LIN {X 0,Y 469.729,Z 273.756,A -85,B 0,C 180,E1 -7607.149,E2 -7607.149} C_VEL
LIN {X 0,Y 469.923,Z 277.249,A -85,B 0,C 180,E1 -7608.848,E2 -7608.848} C_VEL
LIN {X 0,Y 469.592,Z 283.298,A -85,B 0,C 180,E1 -7611.619,E2 -7611.619} C_VEL
LIN {X 0,Y 469.198,Z 289.323,A -85,B 0,C 180,E1 -7614.255,E2 -7614.255} C_VEL
LIN {X 0,Y 468.777,Z 296.664,A -85,B 0,C 180,E1 -7617.335,E2 -7617.335} C_VEL
LIN {X 0,Y 468.436,Z 304.481,A -85,B 0,C 180,E1 -7620.479,E2 -7620.479} C_VEL
LIN {X 0,Y 468.052,Z 312.815,A -85,B 0,C 180,E1 -7623.707,E2 -7623.707} C_VEL
LIN {X 0,Y 467.727,Z 321.729,A -85,B 0,C 180,E1 -7627.003,E2 -7627.003} C_VEL
LIN {X 0,Y 467.618,Z 324.914,A -85,B 0,C 180,E1 -7628.178,E2 -7628.178} C_VEL
LIN {X 0,Y 472.483,Z 344.192,A -85,B 0,C 180,E1 -7628.855,E2 -7628.855} C_VEL
LIN {X 0,Y 473.831,Z 350.735,A -85,B 0,C 180,E1 -7629.122,E2 -7629.122} C_VEL
LIN {X 0,Y 473.198,Z 365.39,A -85,B 0,C 180,E1 -7629.679,E2 -7629.679} C_VEL
LIN {X 0,Y 472.423,Z 380.522,A -85,B 0,C 180,E1 -7630.444,E2 -7630.444} C_VEL
LIN {X 0,Y 471.631,Z 394.097,A -85,B 0,C 180,E1 -7631.314,E2 -7631.314} C_VEL
LIN {X 0,Y 470.815,Z 406.65,A -85,B 0,C 180,E1 -7632.293,E2 -7632.293} C_VEL
LIN {X 0,Y 469.962,Z 419.312,A -85,B 0,C 180,E1 -7633.493,E2 -7633.493} C_VEL
LIN {X 0,Y 469.169,Z 430.767,A -85,B 0,C 180,E1 -7634.803,E2 -7634.803} C_VEL
LIN {X 0,Y 468.498,Z 440.435,A -85,B 0,C 180,E1 -7636.112,E2 -7636.112} C_VEL
LIN {X 0,Y 467.896,Z 449.138,A -85,B 0,C 180,E1 -7637.508,E2 -7637.508} C_VEL
LIN {X 0,Y 467.494,Z 457.77,A -85,B 0,C 180,E1 -7639.169,E2 -7639.169} C_VEL
LIN {X 0,Y 467.07,Z 465.123,A -85,B 0,C 180,E1 -7640.909,E2 -7640.909} C_VEL
LIN {X 0,Y 466.83,Z 470.949,A -85,B 0,C 180,E1 -7642.648,E2 -7642.648} C_VEL
LIN {X 0,Y 466.753,Z 474.383,A -85,B 0,C 180,E1 -7643.95,E2 -7643.95} C_VEL
LIN {X 0,Y 466.619,Z 477.892,A -85,B 0,C 180,E1 -7645.681,E2 -7645.681} C_VEL
LIN {X 0,Y 466.638,Z 480.197,A -85,B 0,C 180,E1 -7647.41,E2 -7647.41} C_VEL
LIN {X 0,Y 466.586,Z 481.352,A -85,B 0,C 180,E1 -7649.137,E2 -7649.137} C_VEL
LIN {X 0,Y 466.586,Z 481.35,A -85,B 0,C 180,E1 -7650.863,E2 -7650.863} C_VEL
LIN {X 0,Y 466.638,Z 480.191,A -85,B 0,C 180,E1 -7652.59,E2 -7652.59} C_VEL
LIN {X 0,Y 466.619,Z 477.886,A -85,B 0,C 180,E1 -7654.319,E2 -7654.319} C_VEL
LIN {X 0,Y 466.768,Z 474.383,A -85,B 0,C 180,E1 -7656.05,E2 -7656.05} C_VEL
LIN {X 0,Y 466.896,Z 469.596,A -85,B 0,C 180,E1 -7657.786,E2 -7657.786} C_VEL
LIN {X 0,Y 467.133,Z 463.399,A -85,B 0,C 180,E1 -7659.526,E2 -7659.526} C_VEL
LIN {X 0,Y 467.614,Z 455.624,A -85,B 0,C 180,E1 -7661.267,E2 -7661.267} C_VEL
LIN {X 0,Y 468.03,Z 447.084,A -85,B 0,C 180,E1 -7662.838,E2 -7662.838} C_VEL
LIN {X 0,Y 468.71,Z 437.348,A -85,B 0,C 180,E1 -7664.324,E2 -7664.324} C_VEL
LIN {X 0,Y 469.341,Z 427.143,A -85,B 0,C 180,E1 -7665.637,E2 -7665.637} C_VEL
LIN {X 0,Y 470.179,Z 415.078,A -85,B 0,C 180,E1 -7666.935,E2 -7666.935} C_VEL
LIN {X 0,Y 471.028,Z 402.621,A -85,B 0,C 180,E1 -7668.035,E2 -7668.035} C_VEL
LIN {X 0,Y 471.897,Z 389.15,A -85,B 0,C 180,E1 -7669.013,E2 -7669.013} C_VEL
LIN {X 0,Y 472.698,Z 375.343,A -85,B 0,C 180,E1 -7669.827,E2 -7669.827} C_VEL
LIN {X 0,Y 473.369,Z 360.123,A -85,B 0,C 180,E1 -7670.532,E2 -7670.532} C_VEL
LIN {X 0,Y 473.644,Z 349.558,A -85,B 0,C 180,E1 -7670.919,E2 -7670.919} C_VEL
LIN {X 0,Y 469.716,Z 332.966,A -85,B 0,C 180,E1 -7671.556,E2 -7671.556} C_VEL
LIN {X 0,Y 467.579,Z 324.175,A -85,B 0,C 180,E1 -7671.844,E2 -7671.844} C_VEL
LIN {X 0,Y 467.838,Z 314.394,A -85,B 0,C 180,E1 -7675.275,E2 -7675.275} C_VEL
LIN {X 0,Y 468.108,Z 306.24,A -85,B 0,C 180,E1 -7678.225,E2 -7678.225} C_VEL
LIN {X 0,Y 468.385,Z 298.351,A -85,B 0,C 180,E1 -7681.211,E2 -7681.211} C_VEL
LIN {X 0,Y 468.622,Z 292.205,A -85,B 0,C 180,E1 -7683.704,E2 -7683.704} C_VEL
LIN {X 0,Y 469.09,Z 285.23,A -85,B 0,C 180,E1 -7686.819,E2 -7686.819} C_VEL
LIN {X 0,Y 469.452,Z 281.021,A -85,B 0,C 180,E1 -7688.96,E2 -7688.96} C_VEL
LIN {X 0,Y 469.801,Z 277.325,A -85,B 0,C 180,E1 -7691.164,E2 -7691.164} C_VEL
LIN {X 0,Y 469.823,Z 275.034,A -85,B 0,C 180,E1 -7692.863,E2 -7692.863} C_VEL
LIN {X 0,Y 469.444,Z 272.713,A -85,B 0,C 180,E1 -7695.281,E2 -7695.281} C_VEL
LIN {X 0,Y 469.093,Z 271.43,A -85,B 0,C 180,E1 -7697.609,E2 -7697.609} C_VEL
LIN {X 0,Y 468.597,Z 271.032,A -85,B 0,C 180,E1 -7699.898,E2 -7699.898} C_VEL
LIN {X 0,Y 468.189,Z 271.444,A -85,B 0,C 180,E1 -7703.099,E2 -7703.099} C_VEL
LIN {X 0,Y 467.827,Z 272.613,A -85,B 0,C 180,E1 -7706.232,E2 -7706.232} C_VEL
LIN {X 0,Y 467.602,Z 274.182,A -85,B 0,C 180,E1 -7709.269,E2 -7709.269} C_VEL
LIN {X 0,Y 467.434,Z 276.177,A -85,B 0,C 180,E1 -7712.509,E2 -7712.509} C_VEL
LIN {X 0,Y 467.341,Z 277.655,A -85,B 0,C 180,E1 -7714.672,E2 -7714.672} C_VEL
LIN {X 0,Y 472.477,Z 293.108,A -85,B 0,C 180,E1 -7715.363,E2 -7715.363} C_VEL
LIN {X 0,Y 473.121,Z 296.754,A -85,B 0,C 180,E1 -7715.523,E2 -7715.523} C_VEL
LIN {X 0,Y 472.61,Z 311.746,A -85,B 0,C 180,E1 -7716.13,E2 -7716.13} C_VEL
LIN {X 0,Y 471.958,Z 326.057,A -85,B 0,C 180,E1 -7716.874,E2 -7716.874} C_VEL
LIN {X 0,Y 471.281,Z 339.483,A -85,B 0,C 180,E1 -7717.746,E2 -7717.746} C_VEL
LIN {X 0,Y 470.652,Z 351.07,A -85,B 0,C 180,E1 -7718.655,E2 -7718.655} C_VEL
LIN {X 0,Y 469.879,Z 364.056,A -85,B 0,C 180,E1 -7719.879,E2 -7719.879} C_VEL
LIN {X 0,Y 469.205,Z 375.809,A -85,B 0,C 180,E1 -7721.214,E2 -7721.214} C_VEL
LIN {X 0,Y 468.589,Z 385.608,A -85,B 0,C 180,E1 -7722.545,E2 -7722.545} C_VEL
LIN {X 0,Y 468.037,Z 395.102,A -85,B 0,C 180,E1 -7724.092,E2 -7724.092} C_VEL
LIN {X 0,Y 467.622,Z 402.939,A -85,B 0,C 180,E1 -7725.642,E2 -7725.642} C_VEL
LIN {X 0,Y 467.278,Z 410.166,A -85,B 0,C 180,E1 -7727.404,E2 -7727.404} C_VEL
LIN {X 0,Y 467.044,Z 415.784,A -85,B 0,C 180,E1 -7729.158,E2 -7729.158} C_VEL
LIN {X 0,Y 466.851,Z 419.086,A -85,B 0,C 180,E1 -7730.468,E2 -7730.468} C_VEL
LIN {X 0,Y 466.794,Z 422.271,A -85,B 0,C 180,E1 -7732.212,E2 -7732.212} C_VEL
LIN {X 0,Y 466.795,Z 424.199,A -85,B 0,C 180,E1 -7733.951,E2 -7733.951} C_VEL
LIN {X 0,Y 466.728,Z 424.95,A -85,B 0,C 180,E1 -7735.682,E2 -7735.682} C_VEL
LIN {X 0,Y 466.782,Z 424.534,A -85,B 0,C 180,E1 -7737.411,E2 -7737.411} C_VEL
LIN {X 0,Y 466.625,Z 422.981,A -85,B 0,C 180,E1 -7739.137,E2 -7739.137} C_VEL
LIN {X 0,Y 466.648,Z 420.238,A -85,B 0,C 180,E1 -7740.863,E2 -7740.863} C_VEL
LIN {X 0,Y 466.881,Z 416.228,A -85,B 0,C 180,E1 -7742.589,E2 -7742.589} C_VEL
LIN {X 0,Y 467.22,Z 410.87,A -85,B 0,C 180,E1 -7744.314,E2 -7744.314} C_VEL
LIN {X 0,Y 467.375,Z 404.075,A -85,B 0,C 180,E1 -7746.042,E2 -7746.042} C_VEL
LIN {X 0,Y 467.914,Z 395.592,A -85,B 0,C 180,E1 -7747.769,E2 -7747.769} C_VEL
LIN {X 0,Y 468.452,Z 386.549,A -85,B 0,C 180,E1 -7749.281,E2 -7749.281} C_VEL
LIN {X 0,Y 469.134,Z 375.671,A -85,B 0,C 180,E1 -7750.793,E2 -7750.793} C_VEL
LIN {X 0,Y 469.839,Z 364.496,A -85,B 0,C 180,E1 -7752.088,E2 -7752.088} C_VEL
LIN {X 0,Y 470.568,Z 352.274,A -85,B 0,C 180,E1 -7753.275,E2 -7753.275} C_VEL
LIN {X 0,Y 471.254,Z 339.027,A -85,B 0,C 180,E1 -7754.346,E2 -7754.346} C_VEL
LIN {X 0,Y 471.989,Z 325.833,A -85,B 0,C 180,E1 -7755.215,E2 -7755.215} C_VEL
LIN {X 0,Y 472.684,Z 310.816,A -85,B 0,C 180,E1 -7756.009,E2 -7756.009} C_VEL
LIN {X 0,Y 473.121,Z 295.089,A -85,B 0,C 180,E1 -7756.644,E2 -7756.644} C_VEL
LIN {X 0,Y 468.818,Z 279.993,A -85,B 0,C 180,E1 -7757.279,E2 -7757.279} C_VEL
LIN {X 0,Y 466.857,Z 273.316,A -85,B 0,C 180,E1 -7757.523,E2 -7757.523} C_VEL
LIN {X 0,Y 466.872,Z 270.616,A -85,B 0,C 180,E1 -7760.257,E2 -7760.257} C_VEL
LIN {X 0,Y 466.934,Z 267.582,A -85,B 0,C 180,E1 -7763.344,E2 -7763.344} C_VEL
LIN {X 0,Y 466.986,Z 265.148,A -85,B 0,C 180,E1 -7765.877,E2 -7765.877} C_VEL
LIN {X 0,Y 467.008,Z 262.347,A -85,B 0,C 180,E1 -7768.788,E2 -7768.788} C_VEL
LIN {X 0,Y 466.989,Z 261.962,A -85,B 0,C 180,E1 -7769.205,E2 -7769.205} C_VEL
LIN {X 0,Y 467.278,Z 261.908,A -85,B 0,C 180,E1 -7771.764,E2 -7771.764} C_VEL
LIN {X 0,Y 467.535,Z 261.872,A -85,B 0,C 180,E1 -7774.835,E2 -7774.835} C_VEL
LIN {X 0,Y 467.566,Z 261.867,A -85,B 0,C 180,E1 -7778.045,E2 -7778.045} C_VEL
LIN {X 0,Y 467.578,Z 261.868,A -85,B 0,C 180,E1 -7781.276,E2 -7781.276} C_VEL
LIN {X 0,Y 467.549,Z 261.868,A -85,B 0,C 180,E1 -7783.82,E2 -7783.82} C_VEL
LIN {X 0,Y 467.558,Z 261.87,A -85,B 0,C 180,E1 -7786.255,E2 -7786.255} C_VEL
LIN {X 0,Y 467.582,Z 261.867,A -85,B 0,C 180,E1 -7788.723,E2 -7788.723} C_VEL
LIN {X 0,Y 467.568,Z 261.867,A -85,B 0,C 180,E1 -7791.955,E2 -7791.955} C_VEL
LIN {X 0,Y 467.562,Z 261.871,A -85,B 0,C 180,E1 -7795.167,E2 -7795.167} C_VEL
LIN {X 0,Y 467.586,Z 261.866,A -85,B 0,C 180,E1 -7798.26,E2 -7798.26} C_VEL
LIN {X 0,Y 467.579,Z 261.868,A -85,B 0,C 180,E1 -7801.25,E2 -7801.25} C_VEL
LIN {X 0,Y 467.59,Z 261.865,A -85,B 0,C 180,E1 -7804.159,E2 -7804.159} C_VEL
LIN {X 0,Y 467.579,Z 261.867,A -85,B 0,C 180,E1 -7806.996,E2 -7806.996} C_VEL
LIN {X 0,Y 467.609,Z 261.862,A -85,B 0,C 180,E1 -7809.599,E2 -7809.599} C_VEL
LIN {X 0,Y 466.981,Z 261.943,A -85,B 0,C 180,E1 -7810.318,E2 -7810.318} C_VEL
LIN {X 0,Y 464.118,Z 262.299,A -85,B 0,C 180,E1 -7811.485,E2 -7811.485} C_VEL
LIN {X 0,Y 461.677,Z 262.603,A -85,B 0,C 180,E1 -7812.426,E2 -7812.426} C_VEL
LIN {X 0,Y 460.64,Z 262.731,A -85,B 0,C 180,E1 -7813.154,E2 -7813.154} C_VEL
LIN {X 0,Y 460.563,Z 262.74,A -85,B 0,C 180,E1 -7813.4,E2 -7813.4} C_VEL
LIN {X 0,Y 460.555,Z 262.742,A -85,B 0,C 180,E1 -7815.868,E2 -7815.868} C_VEL
LIN {X 0,Y 460.613,Z 262.734,A -85,B 0,C 180,E1 -7818.559,E2 -7818.559} C_VEL
LIN {X 0,Y 460.67,Z 262.728,A -85,B 0,C 180,E1 -7822.108,E2 -7822.108} C_VEL
LIN {X 0,Y 460.68,Z 262.724,A -85,B 0,C 180,E1 -7824.748,E2 -7824.748} C_VEL
LIN {X 0,Y 460.795,Z 262.713,A -85,B 0,C 180,E1 -7827.377,E2 -7827.377} C_VEL
LIN {X 0,Y 460.853,Z 262.706,A -85,B 0,C 180,E1 -7830,E2 -7830} C_VEL
LIN {X 0,Y 460.795,Z 262.71,A -85,B 0,C 180,E1 -7832.623,E2 -7832.623} C_VEL
LIN {X 0,Y 460.69,Z 262.727,A -85,B 0,C 180,E1 -7836.13,E2 -7836.13} C_VEL
LIN {X 0,Y 460.622,Z 262.731,A -85,B 0,C 180,E1 -7838.776,E2 -7838.776} C_VEL
LIN {X 0,Y 460.617,Z 262.735,A -85,B 0,C 180,E1 -7842.445,E2 -7842.445} C_VEL
LIN {X 0,Y 460.604,Z 262.735,A -85,B 0,C 180,E1 -7845.998,E2 -7845.998} C_VEL
LIN {X 0,Y 460.572,Z 262.74,A -85,B 0,C 180,E1 -7849.616,E2 -7849.616} C_VEL
LIN {X 0,Y 460.514,Z 262.744,A -85,B 0,C 180,E1 -7852.429,E2 -7852.429} C_VEL
LIN {X 0,Y 460.572,Z 262.741,A -85,B 0,C 180,E1 -7855.802,E2 -7855.802} C_VEL
LIN {X 0,Y 460.554,Z 262.741,A -85,B 0,C 180,E1 -7858.233,E2 -7858.233} C_VEL
LIN {X 0,Y 460.523,Z 262.746,A -85,B 0,C 180,E1 -7861.283,E2 -7861.283} C_VEL
LIN {X 0,Y 460.534,Z 262.744,A -85,B 0,C 180,E1 -7864.505,E2 -7864.505} C_VEL
LIN {X 0,Y 460.502,Z 262.748,A -85,B 0,C 180,E1 -7867.623,E2 -7867.623} C_VEL
LIN {X 0,Y 460.519,Z 262.747,A -85,B 0,C 180,E1 -7871.013,E2 -7871.013} C_VEL
LIN {X 0,Y 460.515,Z 262.748,A -85,B 0,C 180,E1 -7874.589,E2 -7874.589} C_VEL
LIN {X 0,Y 460.527,Z 262.745,A -85,B 0,C 180,E1 -7877.819,E2 -7877.819} C_VEL
LIN {X 0,Y 460.549,Z 262.742,A -85,B 0,C 180,E1 -7881.102,E2 -7881.102} C_VEL
LIN {X 0,Y 460.512,Z 262.747,A -85,B 0,C 180,E1 -7884.554,E2 -7884.554} C_VEL
LIN {X 0,Y 460.534,Z 262.743,A -85,B 0,C 180,E1 -7887.716,E2 -7887.716} C_VEL
LIN {X 0,Y 460.544,Z 262.744,A -85,B 0,C 180,E1 -7890.769,E2 -7890.769} C_VEL
LIN {X 0,Y 460.547,Z 262.74,A -85,B 0,C 180,E1 -7893.733,E2 -7893.733} C_VEL
LIN {X 0,Y 460.549,Z 262.743,A -85,B 0,C 180,E1 -7896.624,E2 -7896.624} C_VEL
LIN {X 0,Y 460.555,Z 262.74,A -85,B 0,C 180,E1 -7899.453,E2 -7899.453} C_VEL
LIN {X 0,Y 460.552,Z 262.744,A -85,B 0,C 180,E1 -7902.23,E2 -7902.23} C_VEL
LIN {X 0,Y 460.567,Z 262.741,A -85,B 0,C 180,E1 -7904.965,E2 -7904.965} C_VEL
LIN {X 0,Y 460.616,Z 262.734,A -85,B 0,C 180,E1 -7908.559,E2 -7908.559} C_VEL
LIN {X 0,Y 460.623,Z 262.733,A -85,B 0,C 180,E1 -7911.224,E2 -7911.224} C_VEL
LIN {X 0,Y 460.675,Z 262.727,A -85,B 0,C 180,E1 -7913.869,E2 -7913.869} C_VEL
LIN {X 0,Y 460.797,Z 262.713,A -85,B 0,C 180,E1 -7917.377,E2 -7917.377} C_VEL
LIN {X 0,Y 460.853,Z 262.706,A -85,B 0,C 180,E1 -7920,E2 -7920} C_VEL
LIN {X 0,Y 460.804,Z 262.71,A -85,B 0,C 180,E1 -7922.622,E2 -7922.622} C_VEL
LIN {X 0,Y 460.687,Z 262.728,A -85,B 0,C 180,E1 -7926.13,E2 -7926.13} C_VEL
LIN {X 0,Y 460.614,Z 262.733,A -85,B 0,C 180,E1 -7928.776,E2 -7928.776} C_VEL
LIN {X 0,Y 460.618,Z 262.734,A -85,B 0,C 180,E1 -7932.445,E2 -7932.445} C_VEL
LIN {X 0,Y 460.604,Z 262.735,A -85,B 0,C 180,E1 -7935.997,E2 -7935.997} C_VEL
LIN {X 0,Y 460.572,Z 262.741,A -85,B 0,C 180,E1 -7939.615,E2 -7939.615} C_VEL
LIN {X 0,Y 460.514,Z 262.745,A -85,B 0,C 180,E1 -7942.428,E2 -7942.428} C_VEL
LIN {X 0,Y 460.551,Z 262.744,A -85,B 0,C 180,E1 -7945.796,E2 -7945.796} C_VEL
LIN {X 0,Y 460.517,Z 262.744,A -85,B 0,C 180,E1 -7948.235,E2 -7948.235} C_VEL
LIN {X 0,Y 460.522,Z 262.746,A -85,B 0,C 180,E1 -7951.282,E2 -7951.282} C_VEL
LIN {X 0,Y 460.533,Z 262.744,A -85,B 0,C 180,E1 -7954.505,E2 -7954.505} C_VEL
LIN {X 0,Y 460.503,Z 262.746,A -85,B 0,C 180,E1 -7957.623,E2 -7957.623} C_VEL
LIN {X 0,Y 460.557,Z 262.915,A -85,B 0,C 180,E1 -7960.393,E2 -7960.393} C_VEL
LIN {X 0,Y 461.469,Z 267.969,A -85,B 0,C 180,E1 -7963.262,E2 -7963.262} C_VEL
LIN {X 0,Y 462.516,Z 273.431,A -85,B 0,C 180,E1 -7966.2,E2 -7966.2} C_VEL
LIN {X 0,Y 462.968,Z 277.166,A -85,B 0,C 180,E1 -7968.092,E2 -7968.092} C_VEL
LIN {X 0,Y 462.775,Z 281.979,A -85,B 0,C 180,E1 -7970.369,E2 -7970.369} C_VEL
LIN {X 0,Y 462.348,Z 289.228,A -85,B 0,C 180,E1 -7973.642,E2 -7973.642} C_VEL
LIN {X 0,Y 461.867,Z 296.621,A -85,B 0,C 180,E1 -7976.815,E2 -7976.815} C_VEL
LIN {X 0,Y 461.448,Z 304.97,A -85,B 0,C 180,E1 -7980.242,E2 -7980.242} C_VEL
LIN {X 0,Y 461.065,Z 312.637,A -85,B 0,C 180,E1 -7983.277,E2 -7983.277} C_VEL
LIN {X 0,Y 460.696,Z 321.458,A -85,B 0,C 180,E1 -7986.632,E2 -7986.632} C_VEL
LIN {X 0,Y 460.593,Z 324.594,A -85,B 0,C 180,E1 -7987.808,E2 -7987.808} C_VEL
LIN {X 0,Y 465.546,Z 344.217,A -85,B 0,C 180,E1 -7988.53,E2 -7988.53} C_VEL
LIN {X 0,Y 467.098,Z 351.971,A -85,B 0,C 180,E1 -7988.86,E2 -7988.86} C_VEL
LIN {X 0,Y 466.496,Z 365.604,A -85,B 0,C 180,E1 -7989.399,E2 -7989.399} C_VEL
LIN {X 0,Y 465.674,Z 380.141,A -85,B 0,C 180,E1 -7990.149,E2 -7990.149} C_VEL
LIN {X 0,Y 464.826,Z 393.687,A -85,B 0,C 180,E1 -7991.03,E2 -7991.03} C_VEL
LIN {X 0,Y 463.889,Z 407.452,A -85,B 0,C 180,E1 -7992.134,E2 -7992.134} C_VEL
LIN {X 0,Y 462.997,Z 419.97,A -85,B 0,C 180,E1 -7993.351,E2 -7993.351} C_VEL
LIN {X 0,Y 462.24,Z 430.537,A -85,B 0,C 180,E1 -7994.569,E2 -7994.569} C_VEL
LIN {X 0,Y 461.537,Z 440.328,A -85,B 0,C 180,E1 -7995.898,E2 -7995.898} C_VEL
LIN {X 0,Y 460.882,Z 449.651,A -85,B 0,C 180,E1 -7997.405,E2 -7997.405} C_VEL
LIN {X 0,Y 460.482,Z 457.77,A -85,B 0,C 180,E1 -7999.002,E2 -7999.002} C_VEL
LIN {X 0,Y 460.008,Z 465.124,A -85,B 0,C 180,E1 -8000.769,E2 -8000.769} C_VEL
LIN {X 0,Y 459.775,Z 470.95,A -85,B 0,C 180,E1 -8002.534,E2 -8002.534} C_VEL
LIN {X 0,Y 459.654,Z 474.382,A -85,B 0,C 180,E1 -8003.856,E2 -8003.856} C_VEL
LIN {X 0,Y 459.538,Z 477.892,A -85,B 0,C 180,E1 -8005.614,E2 -8005.614} C_VEL
LIN {X 0,Y 459.56,Z 480.197,A -85,B 0,C 180,E1 -8007.37,E2 -8007.37} C_VEL
LIN {X 0,Y 459.491,Z 481.352,A -85,B 0,C 180,E1 -8009.124,E2 -8009.124} C_VEL
LIN {X 0,Y 459.491,Z 481.35,A -85,B 0,C 180,E1 -8010.876,E2 -8010.876} C_VEL
LIN {X 0,Y 459.56,Z 480.191,A -85,B 0,C 180,E1 -8012.63,E2 -8012.63} C_VEL
LIN {X 0,Y 459.538,Z 477.886,A -85,B 0,C 180,E1 -8014.386,E2 -8014.386} C_VEL
LIN {X 0,Y 459.696,Z 474.383,A -85,B 0,C 180,E1 -8016.143,E2 -8016.143} C_VEL
LIN {X 0,Y 459.826,Z 469.595,A -85,B 0,C 180,E1 -8017.907,E2 -8017.907} C_VEL
LIN {X 0,Y 460.09,Z 463.397,A -85,B 0,C 180,E1 -8019.673,E2 -8019.673} C_VEL
LIN {X 0,Y 460.609,Z 455.621,A -85,B 0,C 180,E1 -8021.441,E2 -8021.441} C_VEL
LIN {X 0,Y 461.034,Z 447.195,A -85,B 0,C 180,E1 -8023.014,E2 -8023.014} C_VEL
LIN {X 0,Y 461.749,Z 437.152,A -85,B 0,C 180,E1 -8024.545,E2 -8024.545} C_VEL
LIN {X 0,Y 462.434,Z 426.739,A -85,B 0,C 180,E1 -8025.876,E2 -8025.876} C_VEL
LIN {X 0,Y 463.221,Z 415.491,A -85,B 0,C 180,E1 -8027.092,E2 -8027.092} C_VEL
LIN {X 0,Y 464.096,Z 403.283,A -85,B 0,C 180,E1 -8028.2,E2 -8028.2} C_VEL
LIN {X 0,Y 465.003,Z 390.115,A -85,B 0,C 180,E1 -8029.192,E2 -8029.192} C_VEL
LIN {X 0,Y 465.922,Z 375.728,A -85,B 0,C 180,E1 -8030.07,E2 -8030.07} C_VEL
LIN {X 0,Y 466.669,Z 360.221,A -85,B 0,C 180,E1 -8030.813,E2 -8030.813} C_VEL
LIN {X 0,Y 466.883,Z 350.717,A -85,B 0,C 180,E1 -8031.179,E2 -8031.179} C_VEL
LIN {X 0,Y 463.094,Z 334.414,A -85,B 0,C 180,E1 -8031.846,E2 -8031.846} C_VEL
LIN {X 0,Y 460.522,Z 323.542,A -85,B 0,C 180,E1 -8032.224,E2 -8032.224} C_VEL
LIN {X 0,Y 460.849,Z 313.364,A -85,B 0,C 180,E1 -8035.874,E2 -8035.874} C_VEL
LIN {X 0,Y 461.149,Z 304.471,A -85,B 0,C 180,E1 -8039.189,E2 -8039.189} C_VEL
LIN {X 0,Y 461.373,Z 298.703,A -85,B 0,C 180,E1 -8041.457,E2 -8041.457} C_VEL
LIN {X 0,Y 461.677,Z 291.983,A -85,B 0,C 180,E1 -8044.281,E2 -8044.281} C_VEL
LIN {X 0,Y 462.12,Z 286.291,A -85,B 0,C 180,E1 -8046.922,E2 -8046.922} C_VEL
LIN {X 0,Y 462.58,Z 281.19,A -85,B 0,C 180,E1 -8049.651,E2 -8049.651} C_VEL
LIN {X 0,Y 462.895,Z 277.691,A -85,B 0,C 180,E1 -8051.931,E2 -8051.931} C_VEL
LIN {X 0,Y 462.838,Z 276.133,A -85,B 0,C 180,E1 -8053.209,E2 -8053.209} C_VEL
LIN {X 0,Y 462.477,Z 273.958,A -85,B 0,C 180,E1 -8055.651,E2 -8055.651} C_VEL
LIN {X 0,Y 462.02,Z 272.741,A -85,B 0,C 180,E1 -8058.191,E2 -8058.191} C_VEL
LIN {X 0,Y 461.401,Z 272.491,A -85,B 0,C 180,E1 -8061.354,E2 -8061.354} C_VEL
LIN {X 0,Y 461.079,Z 272.988,A -85,B 0,C 180,E1 -8063.887,E2 -8063.887} C_VEL
LIN {X 0,Y 460.755,Z 274.196,A -85,B 0,C 180,E1 -8067.028,E2 -8067.028} C_VEL
LIN {X 0,Y 460.563,Z 275.601,A -85,B 0,C 180,E1 -8069.764,E2 -8069.764} C_VEL
LIN {X 0,Y 460.383,Z 277.413,A -85,B 0,C 180,E1 -8072.744,E2 -8072.744} C_VEL
LIN {X 0,Y 460.297,Z 278.45,A -85,B 0,C 180,E1 -8074.3,E2 -8074.3} C_VEL
LIN {X 0,Y 465.295,Z 292.834,A -85,B 0,C 180,E1 -8074.995,E2 -8074.995} C_VEL
LIN {X 0,Y 466.482,Z 297.88,A -85,B 0,C 180,E1 -8075.239,E2 -8075.239} C_VEL
LIN {X 0,Y 465.943,Z 312.754,A -85,B 0,C 180,E1 -8075.857,E2 -8075.857} C_VEL
LIN {X 0,Y 465.234,Z 327.316,A -85,B 0,C 180,E1 -8076.638,E2 -8076.638} C_VEL
LIN {X 0,Y 464.512,Z 340.216,A -85,B 0,C 180,E1 -8077.499,E2 -8077.499} C_VEL
LIN {X 0,Y 463.774,Z 353.311,A -85,B 0,C 180,E1 -8078.556,E2 -8078.556} C_VEL
LIN {X 0,Y 463.011,Z 365.053,A -85,B 0,C 180,E1 -8079.695,E2 -8079.695} C_VEL
LIN {X 0,Y 462.352,Z 375.706,A -85,B 0,C 180,E1 -8080.925,E2 -8080.925} C_VEL
LIN {X 0,Y 461.693,Z 385.59,A -85,B 0,C 180,E1 -8082.275,E2 -8082.275} C_VEL
LIN {X 0,Y 461.133,Z 394.797,A -85,B 0,C 180,E1 -8083.775,E2 -8083.775} C_VEL
LIN {X 0,Y 460.633,Z 403.125,A -85,B 0,C 180,E1 -8085.419,E2 -8085.419} C_VEL
LIN {X 0,Y 460.263,Z 410.415,A -85,B 0,C 180,E1 -8087.208,E2 -8087.208} C_VEL
LIN {X 0,Y 459.993,Z 416.088,A -85,B 0,C 180,E1 -8088.99,E2 -8088.99} C_VEL
LIN {X 0,Y 459.785,Z 419.432,A -85,B 0,C 180,E1 -8090.321,E2 -8090.321} C_VEL
LIN {X 0,Y 459.727,Z 422.657,A -85,B 0,C 180,E1 -8092.092,E2 -8092.092} C_VEL
LIN {X 0,Y 459.73,Z 424.63,A -85,B 0,C 180,E1 -8093.857,E2 -8093.857} C_VEL
LIN {X 0,Y 459.64,Z 425.42,A -85,B 0,C 180,E1 -8095.616,E2 -8095.616} C_VEL
LIN {X 0,Y 459.695,Z 425.034,A -85,B 0,C 180,E1 -8097.371,E2 -8097.371} C_VEL
LIN {X 0,Y 459.558,Z 423.501,A -85,B 0,C 180,E1 -8099.124,E2 -8099.124} C_VEL
LIN {X 0,Y 459.58,Z 420.772,A -85,B 0,C 180,E1 -8100.876,E2 -8100.876} C_VEL
LIN {X 0,Y 459.828,Z 416.76,A -85,B 0,C 180,E1 -8102.628,E2 -8102.628} C_VEL
LIN {X 0,Y 460.169,Z 411.41,A -85,B 0,C 180,E1 -8104.38,E2 -8104.38} C_VEL
LIN {X 0,Y 460.333,Z 404.622,A -85,B 0,C 180,E1 -8106.135,E2 -8106.135} C_VEL
LIN {X 0,Y 460.897,Z 396.151,A -85,B 0,C 180,E1 -8107.888,E2 -8107.888} C_VEL
LIN {X 0,Y 461.463,Z 387.112,A -85,B 0,C 180,E1 -8109.423,E2 -8109.423} C_VEL
LIN {X 0,Y 462.177,Z 376.259,A -85,B 0,C 180,E1 -8110.958,E2 -8110.958} C_VEL
LIN {X 0,Y 462.945,Z 365.099,A -85,B 0,C 180,E1 -8112.271,E2 -8112.271} C_VEL
LIN {X 0,Y 463.688,Z 352.911,A -85,B 0,C 180,E1 -8113.476,E2 -8113.476} C_VEL
LIN {X 0,Y 464.451,Z 339.387,A -85,B 0,C 180,E1 -8114.586,E2 -8114.586} C_VEL
LIN {X 0,Y 465.308,Z 324.781,A -85,B 0,C 180,E1 -8115.551,E2 -8115.551} C_VEL
LIN {X 0,Y 465.97,Z 310.54,A -85,B 0,C 180,E1 -8116.303,E2 -8116.303} C_VEL
LIN {X 0,Y 466.382,Z 296.485,A -85,B 0,C 180,E1 -8116.884,E2 -8116.884} C_VEL
LIN {X 0,Y 461.857,Z 280.625,A -85,B 0,C 180,E1 -8117.576,E2 -8117.576} C_VEL
LIN {X 0,Y 459.812,Z 273.697,A -85,B 0,C 180,E1 -8117.828,E2 -8117.828} C_VEL
LIN {X 0,Y 459.821,Z 270.356,A -85,B 0,C 180,E1 -8121.197,E2 -8121.197} C_VEL
LIN {X 0,Y 459.885,Z 267.272,A -85,B 0,C 180,E1 -8124.37,E2 -8124.37} C_VEL
LIN {X 0,Y 459.938,Z 264.479,A -85,B 0,C 180,E1 -8127.285,E2 -8127.285} C_VEL
LIN {X 0,Y 459.969,Z 262.818,A -85,B 0,C 180,E1 -8129.434,E2 -8129.434} C_VEL
LIN {X 0,Y 460.269,Z 262.779,A -85,B 0,C 180,E1 -8132.305,E2 -8132.305} C_VEL
LIN {X 0,Y 460.485,Z 262.751,A -85,B 0,C 180,E1 -8134.496,E2 -8134.496} C_VEL
LIN {X 0,Y 460.502,Z 262.747,A -85,B 0,C 180,E1 -8137.623,E2 -8137.623} C_VEL
LIN {X 0,Y 460.54,Z 262.744,A -85,B 0,C 180,E1 -8140.269,E2 -8140.269} C_VEL
LIN {X 0,Y 460.512,Z 262.747,A -85,B 0,C 180,E1 -8143.374,E2 -8143.374} C_VEL
LIN {X 0,Y 460.502,Z 262.75,A -85,B 0,C 180,E1 -8146.625,E2 -8146.625} C_VEL
LIN {X 0,Y 460.542,Z 262.742,A -85,B 0,C 180,E1 -8149.731,E2 -8149.731} C_VEL
LIN {X 0,Y 460.503,Z 262.751,A -85,B 0,C 180,E1 -8152.524,E2 -8152.524} C_VEL
LIN {X 0,Y 460.54,Z 262.743,A -85,B 0,C 180,E1 -8155.623,E2 -8155.623} C_VEL
LIN {X 0,Y 460.541,Z 262.744,A -85,B 0,C 180,E1 -8158.745,E2 -8158.745} C_VEL
LIN {X 0,Y 460.581,Z 262.738,A -85,B 0,C 180,E1 -8162.255,E2 -8162.255} C_VEL
LIN {X 0,Y 460.532,Z 262.746,A -85,B 0,C 180,E1 -8164.704,E2 -8164.704} C_VEL
LIN {X 0,Y 460.514,Z 262.747,A -85,B 0,C 180,E1 -8167.571,E2 -8167.571} C_VEL
LIN {X 0,Y 460.571,Z 262.742,A -85,B 0,C 180,E1 -8170.384,E2 -8170.384} C_VEL
LIN {X 0,Y 460.563,Z 262.74,A -85,B 0,C 180,E1 -8173.4,E2 -8173.4} C_VEL
LIN {X 0,Y 459.905,Z 262.824,A -85,B 0,C 180,E1 -8174.13,E2 -8174.13} C_VEL
LIN {X 0,Y 457.023,Z 263.182,A -85,B 0,C 180,E1 -8175.315,E2 -8175.315} C_VEL
LIN {X 0,Y 454.603,Z 263.484,A -85,B 0,C 180,E1 -8176.271,E2 -8176.271} C_VEL
LIN {X 0,Y 453.603,Z 263.607,A -85,B 0,C 180,E1 -8177.01,E2 -8177.01} C_VEL
LIN {X 0,Y 453.543,Z 263.613,A -85,B 0,C 180,E1 -8177.26,E2 -8177.26} C_VEL
LIN {X 0,Y 453.574,Z 263.612,A -85,B 0,C 180,E1 -8180.186,E2 -8180.186} C_VEL
LIN {X 0,Y 453.591,Z 263.609,A -85,B 0,C 180,E1 -8182.88,E2 -8182.88} C_VEL
LIN {X 0,Y 453.653,Z 263.6,A -85,B 0,C 180,E1 -8184.667,E2 -8184.667} C_VEL
LIN {X 0,Y 453.739,Z 263.591,A -85,B 0,C 180,E1 -8187.337,E2 -8187.337} C_VEL
LIN {X 0,Y 453.823,Z 263.581,A -85,B 0,C 180,E1 -8190,E2 -8190} C_VEL
LIN {X 0,Y 453.739,Z 263.589,A -85,B 0,C 180,E1 -8192.663,E2 -8192.663} C_VEL
LIN {X 0,Y 453.656,Z 263.604,A -85,B 0,C 180,E1 -8196.226,E2 -8196.226} C_VEL
LIN {X 0,Y 453.588,Z 263.607,A -85,B 0,C 180,E1 -8198.914,E2 -8198.914} C_VEL
LIN {X 0,Y 453.567,Z 263.612,A -85,B 0,C 180,E1 -8202.529,E2 -8202.529} C_VEL
LIN {X 0,Y 453.548,Z 263.613,A -85,B 0,C 180,E1 -8206.196,E2 -8206.196} C_VEL
LIN {X 0,Y 453.521,Z 263.619,A -85,B 0,C 180,E1 -8209.04,E2 -8209.04} C_VEL
LIN {X 0,Y 453.48,Z 263.624,A -85,B 0,C 180,E1 -8211.836,E2 -8211.836} C_VEL
LIN {X 0,Y 453.517,Z 263.619,A -85,B 0,C 180,E1 -8214.734,E2 -8214.734} C_VEL
LIN {X 0,Y 453.535,Z 263.616,A -85,B 0,C 180,E1 -8217.959,E2 -8217.959} C_VEL
LIN {X 0,Y 453.469,Z 263.624,A -85,B 0,C 180,E1 -8221.525,E2 -8221.525} C_VEL
LIN {X 0,Y 453.49,Z 263.621,A -85,B 0,C 180,E1 -8224.777,E2 -8224.777} C_VEL
LIN {X 0,Y 453.461,Z 263.625,A -85,B 0,C 180,E1 -8228.312,E2 -8228.312} C_VEL
LIN {X 0,Y 453.473,Z 263.624,A -85,B 0,C 180,E1 -8230.612,E2 -8230.612} C_VEL
LIN {X 0,Y 453.462,Z 263.624,A -85,B 0,C 180,E1 -8234.222,E2 -8234.222} C_VEL
LIN {X 0,Y 453.467,Z 263.625,A -85,B 0,C 180,E1 -8237.005,E2 -8237.005} C_VEL
LIN {X 0,Y 453.509,Z 263.62,A -85,B 0,C 180,E1 -8240.552,E2 -8240.552} C_VEL
LIN {X 0,Y 453.458,Z 263.626,A -85,B 0,C 180,E1 -8243.917,E2 -8243.917} C_VEL
LIN {X 0,Y 453.483,Z 263.622,A -85,B 0,C 180,E1 -8247.151,E2 -8247.151} C_VEL
LIN {X 0,Y 453.48,Z 263.624,A -85,B 0,C 180,E1 -8250.268,E2 -8250.268} C_VEL
LIN {X 0,Y 453.493,Z 263.619,A -85,B 0,C 180,E1 -8253.293,E2 -8253.293} C_VEL
LIN {X 0,Y 453.501,Z 263.622,A -85,B 0,C 180,E1 -8256.238,E2 -8256.238} C_VEL
LIN {X 0,Y 453.487,Z 263.622,A -85,B 0,C 180,E1 -8259.118,E2 -8259.118} C_VEL
LIN {X 0,Y 453.507,Z 263.621,A -85,B 0,C 180,E1 -8261.944,E2 -8261.944} C_VEL
LIN {X 0,Y 453.543,Z 263.618,A -85,B 0,C 180,E1 -8264.726,E2 -8264.726} C_VEL
LIN {X 0,Y 453.565,Z 263.613,A -85,B 0,C 180,E1 -8268.379,E2 -8268.379} C_VEL
LIN {X 0,Y 453.589,Z 263.609,A -85,B 0,C 180,E1 -8271.086,E2 -8271.086} C_VEL
LIN {X 0,Y 453.642,Z 263.603,A -85,B 0,C 180,E1 -8273.774,E2 -8273.774} C_VEL
LIN {X 0,Y 453.741,Z 263.591,A -85,B 0,C 180,E1 -8277.336,E2 -8277.336} C_VEL
LIN {X 0,Y 453.822,Z 263.582,A -85,B 0,C 180,E1 -8280,E2 -8280} C_VEL
LIN {X 0,Y 453.748,Z 263.589,A -85,B 0,C 180,E1 -8282.663,E2 -8282.663} C_VEL
LIN {X 0,Y 453.652,Z 263.604,A -85,B 0,C 180,E1 -8286.225,E2 -8286.225} C_VEL
LIN {X 0,Y 453.582,Z 263.609,A -85,B 0,C 180,E1 -8288.913,E2 -8288.913} C_VEL
LIN {X 0,Y 453.568,Z 263.612,A -85,B 0,C 180,E1 -8292.529,E2 -8292.529} C_VEL
LIN {X 0,Y 453.548,Z 263.614,A -85,B 0,C 180,E1 -8296.196,E2 -8296.196} C_VEL
LIN {X 0,Y 453.521,Z 263.618,A -85,B 0,C 180,E1 -8299.039,E2 -8299.039} C_VEL
LIN {X 0,Y 453.48,Z 263.623,A -85,B 0,C 180,E1 -8301.836,E2 -8301.836} C_VEL
LIN {X 0,Y 453.503,Z 263.621,A -85,B 0,C 180,E1 -8304.735,E2 -8304.735} C_VEL
LIN {X 0,Y 453.478,Z 263.622,A -85,B 0,C 180,E1 -8307.946,E2 -8307.946} C_VEL
LIN {X 0,Y 453.476,Z 263.625,A -85,B 0,C 180,E1 -8310.759,E2 -8310.759} C_VEL
LIN {X 0,Y 453.478,Z 263.626,A -85,B 0,C 180,E1 -8313.912,E2 -8313.912} C_VEL
LIN {X 0,Y 453.454,Z 263.624,A -85,B 0,C 180,E1 -8317.189,E2 -8317.189} C_VEL
LIN {X 0,Y 453.51,Z 263.697,A -85,B 0,C 180,E1 -8319.88,E2 -8319.88} C_VEL
LIN {X 0,Y 454.413,Z 268.888,A -85,B 0,C 180,E1 -8322.883,E2 -8322.883} C_VEL
LIN {X 0,Y 455.528,Z 274.634,A -85,B 0,C 180,E1 -8326.03,E2 -8326.03} C_VEL
LIN {X 0,Y 455.98,Z 277.892,A -85,B 0,C 180,E1 -8327.716,E2 -8327.716} C_VEL
LIN {X 0,Y 455.944,Z 281.877,A -85,B 0,C 180,E1 -8329.654,E2 -8329.654} C_VEL
LIN {X 0,Y 455.472,Z 289.124,A -85,B 0,C 180,E1 -8333.002,E2 -8333.002} C_VEL
LIN {X 0,Y 454.9,Z 297.195,A -85,B 0,C 180,E1 -8336.54,E2 -8336.54} C_VEL
LIN {X 0,Y 454.445,Z 305.445,A -85,B 0,C 180,E1 -8340.002,E2 -8340.002} C_VEL
LIN {X 0,Y 454.071,Z 312.444,A -85,B 0,C 180,E1 -8342.832,E2 -8342.832} C_VEL
LIN {X 0,Y 453.668,Z 321.188,A -85,B 0,C 180,E1 -8346.248,E2 -8346.248} C_VEL
LIN {X 0,Y 453.571,Z 324.343,A -85,B 0,C 180,E1 -8347.452,E2 -8347.452} C_VEL
LIN {X 0,Y 458.111,Z 342.366,A -85,B 0,C 180,E1 -8348.112,E2 -8348.112} C_VEL
LIN {X 0,Y 460.382,Z 353.364,A -85,B 0,C 180,E1 -8348.598,E2 -8348.598} C_VEL
LIN {X 0,Y 459.734,Z 367.582,A -85,B 0,C 180,E1 -8349.199,E2 -8349.199} C_VEL
LIN {X 0,Y 458.839,Z 381.574,A -85,B 0,C 180,E1 -8349.957,E2 -8349.957} C_VEL
LIN {X 0,Y 457.948,Z 394.753,A -85,B 0,C 180,E1 -8350.85,E2 -8350.85} C_VEL
LIN {X 0,Y 456.967,Z 408.25,A -85,B 0,C 180,E1 -8351.97,E2 -8351.97} C_VEL
LIN {X 0,Y 456.044,Z 420.565,A -85,B 0,C 180,E1 -8353.205,E2 -8353.205} C_VEL
LIN {X 0,Y 455.168,Z 431.824,A -85,B 0,C 180,E1 -8354.553,E2 -8354.553} C_VEL
LIN {X 0,Y 454.337,Z 442.788,A -85,B 0,C 180,E1 -8356.127,E2 -8356.127} C_VEL
LIN {X 0,Y 453.691,Z 451.903,A -85,B 0,C 180,E1 -8357.702,E2 -8357.702} C_VEL
LIN {X 0,Y 453.251,Z 459.496,A -85,B 0,C 180,E1 -8359.276,E2 -8359.276} C_VEL
LIN {X 0,Y 452.886,Z 466.569,A -85,B 0,C 180,E1 -8361.073,E2 -8361.073} C_VEL
LIN {X 0,Y 452.658,Z 472.137,A -85,B 0,C 180,E1 -8362.865,E2 -8362.865} C_VEL
LIN {X 0,Y 452.546,Z 476.291,A -85,B 0,C 180,E1 -8364.653,E2 -8364.653} C_VEL
LIN {X 0,Y 452.438,Z 479.191,A -85,B 0,C 180,E1 -8366.438,E2 -8366.438} C_VEL
LIN {X 0,Y 452.429,Z 480.916,A -85,B 0,C 180,E1 -8368.22,E2 -8368.22} C_VEL
LIN {X 0,Y 452.378,Z 481.5,A -85,B 0,C 180,E1 -8370,E2 -8370} C_VEL
LIN {X 0,Y 452.429,Z 480.912,A -85,B 0,C 180,E1 -8371.78,E2 -8371.78} C_VEL
LIN {X 0,Y 452.438,Z 479.184,A -85,B 0,C 180,E1 -8373.562,E2 -8373.562} C_VEL
LIN {X 0,Y 452.553,Z 476.288,A -85,B 0,C 180,E1 -8375.346,E2 -8375.346} C_VEL
LIN {X 0,Y 452.661,Z 472.141,A -85,B 0,C 180,E1 -8377.135,E2 -8377.135} C_VEL
LIN {X 0,Y 452.886,Z 466.555,A -85,B 0,C 180,E1 -8378.927,E2 -8378.927} C_VEL
LIN {X 0,Y 453.25,Z 459.432,A -85,B 0,C 180,E1 -8380.724,E2 -8380.724} C_VEL
LIN {X 0,Y 453.703,Z 451.79,A -85,B 0,C 180,E1 -8382.298,E2 -8382.298} C_VEL
LIN {X 0,Y 454.309,Z 442.599,A -85,B 0,C 180,E1 -8383.874,E2 -8383.874} C_VEL
LIN {X 0,Y 455.006,Z 433.263,A -85,B 0,C 180,E1 -8385.223,E2 -8385.223} C_VEL
LIN {X 0,Y 455.885,Z 421.186,A -85,B 0,C 180,E1 -8386.686,E2 -8386.686} C_VEL
LIN {X 0,Y 456.835,Z 408.954,A -85,B 0,C 180,E1 -8387.92,E2 -8387.92} C_VEL
LIN {X 0,Y 457.799,Z 395.572,A -85,B 0,C 180,E1 -8389.04,E2 -8389.04} C_VEL
LIN {X 0,Y 458.781,Z 380.796,A -85,B 0,C 180,E1 -8390.045,E2 -8390.045} C_VEL
LIN {X 0,Y 459.742,Z 365.139,A -85,B 0,C 180,E1 -8390.883,E2 -8390.883} C_VEL
LIN {X 0,Y 460.239,Z 352.143,A -85,B 0,C 180,E1 -8391.43,E2 -8391.43} C_VEL
LIN {X 0,Y 456.463,Z 335.601,A -85,B 0,C 180,E1 -8392.149,E2 -8392.149} C_VEL
LIN {X 0,Y 453.46,Z 322.892,A -85,B 0,C 180,E1 -8392.619,E2 -8392.619} C_VEL
LIN {X 0,Y 453.785,Z 313.475,A -85,B 0,C 180,E1 -8396.068,E2 -8396.068} C_VEL
LIN {X 0,Y 454.089,Z 305.338,A -85,B 0,C 180,E1 -8399.179,E2 -8399.179} C_VEL
LIN {X 0,Y 454.406,Z 297.787,A -85,B 0,C 180,E1 -8402.249,E2 -8402.249} C_VEL
LIN {X 0,Y 454.784,Z 291.525,A -85,B 0,C 180,E1 -8405.012,E2 -8405.012} C_VEL
LIN {X 0,Y 455.137,Z 287.364,A -85,B 0,C 180,E1 -8407.029,E2 -8407.029} C_VEL
LIN {X 0,Y 455.598,Z 282.79,A -85,B 0,C 180,E1 -8409.53,E2 -8409.53} C_VEL
LIN {X 0,Y 455.88,Z 279.733,A -85,B 0,C 180,E1 -8411.522,E2 -8411.522} C_VEL
LIN {X 0,Y 455.83,Z 277.267,A -85,B 0,C 180,E1 -8413.561,E2 -8413.561} C_VEL
LIN {X 0,Y 455.478,Z 275.223,A -85,B 0,C 180,E1 -8416.025,E2 -8416.025} C_VEL
LIN {X 0,Y 455.028,Z 274.17,A -85,B 0,C 180,E1 -8418.384,E2 -8418.384} C_VEL
LIN {X 0,Y 454.573,Z 273.861,A -85,B 0,C 180,E1 -8420.663,E2 -8420.663} C_VEL
LIN {X 0,Y 454.086,Z 274.327,A -85,B 0,C 180,E1 -8423.975,E2 -8423.975} C_VEL
LIN {X 0,Y 453.771,Z 275.482,A -85,B 0,C 180,E1 -8427.175,E2 -8427.175} C_VEL
LIN {X 0,Y 453.525,Z 277.041,A -85,B 0,C 180,E1 -8430.272,E2 -8430.272} C_VEL
LIN {X 0,Y 453.444,Z 278.219,A -85,B 0,C 180,E1 -8432.292,E2 -8432.292} C_VEL
LIN {X 0,Y 453.313,Z 279.355,A -85,B 0,C 180,E1 -8433.928,E2 -8433.928} C_VEL
LIN {X 0,Y 458.542,Z 293.82,A -85,B 0,C 180,E1 -8434.667,E2 -8434.667} C_VEL
LIN {X 0,Y 459.89,Z 299.391,A -85,B 0,C 180,E1 -8434.95,E2 -8434.95} C_VEL
LIN {X 0,Y 459.219,Z 315.458,A -85,B 0,C 180,E1 -8435.653,E2 -8435.653} C_VEL
LIN {X 0,Y 458.393,Z 330.46,A -85,B 0,C 180,E1 -8436.508,E2 -8436.508} C_VEL
LIN {X 0,Y 457.571,Z 344.903,A -85,B 0,C 180,E1 -8437.539,E2 -8437.539} C_VEL
LIN {X 0,Y 456.827,Z 356.824,A -85,B 0,C 180,E1 -8438.569,E2 -8438.569} C_VEL
LIN {X 0,Y 456.058,Z 368.368,A -85,B 0,C 180,E1 -8439.76,E2 -8439.76} C_VEL
LIN {X 0,Y 455.298,Z 379.226,A -85,B 0,C 180,E1 -8441.086,E2 -8441.086} C_VEL
LIN {X 0,Y 454.633,Z 388.668,A -85,B 0,C 180,E1 -8442.456,E2 -8442.456} C_VEL
LIN {X 0,Y 454.022,Z 397.827,A -85,B 0,C 180,E1 -8444.052,E2 -8444.052} C_VEL
LIN {X 0,Y 453.567,Z 405.35,A -85,B 0,C 180,E1 -8445.646,E2 -8445.646} C_VEL
LIN {X 0,Y 453.186,Z 412.304,A -85,B 0,C 180,E1 -8447.461,E2 -8447.461} C_VEL
LIN {X 0,Y 452.904,Z 417.66,A -85,B 0,C 180,E1 -8449.268,E2 -8449.268} C_VEL
LIN {X 0,Y 452.691,Z 421.589,A -85,B 0,C 180,E1 -8451.069,E2 -8451.069} C_VEL
LIN {X 0,Y 452.641,Z 424.215,A -85,B 0,C 180,E1 -8452.865,E2 -8452.865} C_VEL
LIN {X 0,Y 452.585,Z 425.626,A -85,B 0,C 180,E1 -8454.654,E2 -8454.654} C_VEL
LIN {X 0,Y 452.613,Z 425.854,A -85,B 0,C 180,E1 -8456.439,E2 -8456.439} C_VEL
LIN {X 0,Y 452.576,Z 424.92,A -85,B 0,C 180,E1 -8458.22,E2 -8458.22} C_VEL
LIN {X 0,Y 452.48,Z 422.817,A -85,B 0,C 180,E1 -8460,E2 -8460} C_VEL
LIN {X 0,Y 452.62,Z 419.46,A -85,B 0,C 180,E1 -8461.78,E2 -8461.78} C_VEL
LIN {X 0,Y 453.006,Z 414.787,A -85,B 0,C 180,E1 -8463.558,E2 -8463.558} C_VEL
LIN {X 0,Y 453.266,Z 408.747,A -85,B 0,C 180,E1 -8465.338,E2 -8465.338} C_VEL
LIN {X 0,Y 453.547,Z 401.656,A -85,B 0,C 180,E1 -8467.012,E2 -8467.012} C_VEL
LIN {X 0,Y 454.126,Z 393.014,A -85,B 0,C 180,E1 -8468.679,E2 -8468.679} C_VEL
LIN {X 0,Y 454.808,Z 383.254,A -85,B 0,C 180,E1 -8470.236,E2 -8470.236} C_VEL
LIN {X 0,Y 455.446,Z 373.296,A -85,B 0,C 180,E1 -8471.572,E2 -8471.572} C_VEL
LIN {X 0,Y 456.316,Z 361.48,A -85,B 0,C 180,E1 -8472.905,E2 -8472.905} C_VEL
LIN {X 0,Y 457.053,Z 349.767,A -85,B 0,C 180,E1 -8474.016,E2 -8474.016} C_VEL
LIN {X 0,Y 457.823,Z 337.16,A -85,B 0,C 180,E1 -8475.017,E2 -8475.017} C_VEL
LIN {X 0,Y 458.624,Z 323.647,A -85,B 0,C 180,E1 -8475.898,E2 -8475.898} C_VEL
LIN {X 0,Y 459.308,Z 310.139,A -85,B 0,C 180,E1 -8476.608,E2 -8476.608} C_VEL
LIN {X 0,Y 459.563,Z 297.601,A -85,B 0,C 180,E1 -8477.141,E2 -8477.141} C_VEL
LIN {X 0,Y 455.283,Z 282.508,A -85,B 0,C 180,E1 -8477.818,E2 -8477.818} C_VEL
LIN {X 0,Y 452.756,Z 274.015,A -85,B 0,C 180,E1 -8478.155,E2 -8478.155} C_VEL
LIN {X 0,Y 452.764,Z 270.886,A -85,B 0,C 180,E1 -8481.353,E2 -8481.353} C_VEL
LIN {X 0,Y 452.853,Z 267.575,A -85,B 0,C 180,E1 -8484.773,E2 -8484.773} C_VEL
LIN {X 0,Y 452.862,Z 264.685,A -85,B 0,C 180,E1 -8487.798,E2 -8487.798} C_VEL
LIN {X 0,Y 452.875,Z 263.792,A -85,B 0,C 180,E1 -8488.756,E2 -8488.756} C_VEL
LIN {X 0,Y 453.171,Z 263.664,A -85,B 0,C 180,E1 -8491.823,E2 -8491.823} C_VEL
LIN {X 0,Y 453.432,Z 263.629,A -85,B 0,C 180,E1 -8494.766,E2 -8494.766} C_VEL
LIN {X 0,Y 453.45,Z 263.625,A -85,B 0,C 180,E1 -8497.772,E2 -8497.772} C_VEL
LIN {X 0,Y 453.497,Z 263.622,A -85,B 0,C 180,E1 -8500.609,E2 -8500.609} C_VEL
LIN {X 0,Y 453.463,Z 263.623,A -85,B 0,C 180,E1 -8504.222,E2 -8504.222} C_VEL
LIN {X 0,Y 453.466,Z 263.625,A -85,B 0,C 180,E1 -8507.005,E2 -8507.005} C_VEL
LIN {X 0,Y 453.498,Z 263.621,A -85,B 0,C 180,E1 -8509.409,E2 -8509.409} C_VEL
LIN {X 0,Y 453.452,Z 263.627,A -85,B 0,C 180,E1 -8512.227,E2 -8512.227} C_VEL
LIN {X 0,Y 453.486,Z 263.624,A -85,B 0,C 180,E1 -8515.224,E2 -8515.224} C_VEL
LIN {X 0,Y 453.469,Z 263.627,A -85,B 0,C 180,E1 -8518.475,E2 -8518.475} C_VEL
LIN {X 0,Y 453.533,Z 263.617,A -85,B 0,C 180,E1 -8522.041,E2 -8522.041} C_VEL
LIN {X 0,Y 453.495,Z 263.62,A -85,B 0,C 180,E1 -8525.264,E2 -8525.264} C_VEL
LIN {X 0,Y 453.484,Z 263.623,A -85,B 0,C 180,E1 -8528.415,E2 -8528.415} C_VEL
LIN {X 0,Y 453.525,Z 263.616,A -85,B 0,C 180,E1 -8531.009,E2 -8531.009} C_VEL
LIN {X 0,Y 453.572,Z 263.614,A -85,B 0,C 180,E1 -8533.88,E2 -8533.88} C_VEL
LIN {X 0,Y 453.543,Z 263.613,A -85,B 0,C 180,E1 -8537.26,E2 -8537.26} C_VEL
LIN {X 0,Y 452.932,Z 263.693,A -85,B 0,C 180,E1 -8538.001,E2 -8538.001} C_VEL
LIN {X 0,Y 450.091,Z 264.046,A -85,B 0,C 180,E1 -8539.204,E2 -8539.204} C_VEL
LIN {X 0,Y 447.658,Z 264.349,A -85,B 0,C 180,E1 -8540.175,E2 -8540.175} C_VEL
LIN {X 0,Y 446.619,Z 264.478,A -85,B 0,C 180,E1 -8540.926,E2 -8540.926} C_VEL
LIN {X 0,Y 446.539,Z 264.487,A -85,B 0,C 180,E1 -8541.18,E2 -8541.18} C_VEL
LIN {X 0,Y 446.613,Z 264.478,A -85,B 0,C 180,E1 -8543.676,E2 -8543.676} C_VEL
LIN {X 0,Y 446.686,Z 264.469,A -85,B 0,C 180,E1 -8547.295,E2 -8547.295} C_VEL
LIN {X 0,Y 446.792,Z 264.457,A -85,B 0,C 180,E1 -8550,E2 -8550} C_VEL
LIN {X 0,Y 446.686,Z 264.468,A -85,B 0,C 180,E1 -8552.705,E2 -8552.705} C_VEL
LIN {X 0,Y 446.624,Z 264.478,A -85,B 0,C 180,E1 -8556.324,E2 -8556.324} C_VEL
LIN {X 0,Y 446.523,Z 264.49,A -85,B 0,C 180,E1 -8559.97,E2 -8559.97} C_VEL
LIN {X 0,Y 446.525,Z 264.489,A -85,B 0,C 180,E1 -8562.73,E2 -8562.73} C_VEL
LIN {X 0,Y 446.492,Z 264.492,A -85,B 0,C 180,E1 -8566.459,E2 -8566.459} C_VEL
LIN {X 0,Y 446.472,Z 264.496,A -85,B 0,C 180,E1 -8569.303,E2 -8569.303} C_VEL
LIN {X 0,Y 446.421,Z 264.5,A -85,B 0,C 180,E1 -8572.2,E2 -8572.2} C_VEL
LIN {X 0,Y 446.461,Z 264.499,A -85,B 0,C 180,E1 -8575.152,E2 -8575.152} C_VEL
LIN {X 0,Y 446.488,Z 264.493,A -85,B 0,C 180,E1 -8578.179,E2 -8578.179} C_VEL
LIN {X 0,Y 446.422,Z 264.502,A -85,B 0,C 180,E1 -8581.775,E2 -8581.775} C_VEL
LIN {X 0,Y 446.432,Z 264.5,A -85,B 0,C 180,E1 -8584.523,E2 -8584.523} C_VEL
LIN {X 0,Y 446.414,Z 264.503,A -85,B 0,C 180,E1 -8588.078,E2 -8588.078} C_VEL
LIN {X 0,Y 446.405,Z 264.506,A -85,B 0,C 180,E1 -8591.394,E2 -8591.394} C_VEL
LIN {X 0,Y 446.454,Z 264.499,A -85,B 0,C 180,E1 -8595.104,E2 -8595.104} C_VEL
LIN {X 0,Y 446.432,Z 264.501,A -85,B 0,C 180,E1 -8598.609,E2 -8598.609} C_VEL
LIN {X 0,Y 446.459,Z 264.498,A -85,B 0,C 180,E1 -8600.974,E2 -8600.974} C_VEL
LIN {X 0,Y 446.422,Z 264.502,A -85,B 0,C 180,E1 -8604.374,E2 -8604.374} C_VEL
LIN {X 0,Y 446.424,Z 264.5,A -85,B 0,C 180,E1 -8607.638,E2 -8607.638} C_VEL
LIN {X 0,Y 446.453,Z 264.499,A -85,B 0,C 180,E1 -8610.791,E2 -8610.791} C_VEL
LIN {X 0,Y 446.465,Z 264.495,A -85,B 0,C 180,E1 -8613.847,E2 -8613.847} C_VEL
LIN {X 0,Y 446.431,Z 264.502,A -85,B 0,C 180,E1 -8616.823,E2 -8616.823} C_VEL
LIN {X 0,Y 446.448,Z 264.497,A -85,B 0,C 180,E1 -8619.737,E2 -8619.737} C_VEL
LIN {X 0,Y 446.46,Z 264.498,A -85,B 0,C 180,E1 -8622.597,E2 -8622.597} C_VEL
LIN {X 0,Y 446.471,Z 264.495,A -85,B 0,C 180,E1 -8625.412,E2 -8625.412} C_VEL
LIN {X 0,Y 446.523,Z 264.492,A -85,B 0,C 180,E1 -8628.193,E2 -8628.193} C_VEL
LIN {X 0,Y 446.537,Z 264.488,A -85,B 0,C 180,E1 -8630.944,E2 -8630.944} C_VEL
LIN {X 0,Y 446.612,Z 264.478,A -85,B 0,C 180,E1 -8633.676,E2 -8633.676} C_VEL
LIN {X 0,Y 446.688,Z 264.469,A -85,B 0,C 180,E1 -8637.294,E2 -8637.294} C_VEL
LIN {X 0,Y 446.792,Z 264.458,A -85,B 0,C 180,E1 -8640,E2 -8640} C_VEL
LIN {X 0,Y 446.695,Z 264.468,A -85,B 0,C 180,E1 -8642.705,E2 -8642.705} C_VEL
LIN {X 0,Y 446.621,Z 264.478,A -85,B 0,C 180,E1 -8646.324,E2 -8646.324} C_VEL
LIN {X 0,Y 446.53,Z 264.488,A -85,B 0,C 180,E1 -8649.055,E2 -8649.055} C_VEL
LIN {X 0,Y 446.525,Z 264.489,A -85,B 0,C 180,E1 -8652.729,E2 -8652.729} C_VEL
LIN {X 0,Y 446.493,Z 264.493,A -85,B 0,C 180,E1 -8656.459,E2 -8656.459} C_VEL
LIN {X 0,Y 446.472,Z 264.496,A -85,B 0,C 180,E1 -8659.303,E2 -8659.303} C_VEL
LIN {X 0,Y 446.421,Z 264.501,A -85,B 0,C 180,E1 -8662.199,E2 -8662.199} C_VEL
LIN {X 0,Y 446.445,Z 264.5,A -85,B 0,C 180,E1 -8665.153,E2 -8665.153} C_VEL
LIN {X 0,Y 446.44,Z 264.497,A -85,B 0,C 180,E1 -8668.182,E2 -8668.182} C_VEL
LIN {X 0,Y 446.417,Z 264.503,A -85,B 0,C 180,E1 -8671.3,E2 -8671.3} C_VEL
LIN {X 0,Y 446.43,Z 264.501,A -85,B 0,C 180,E1 -8674.523,E2 -8674.523} C_VEL
LIN {X 0,Y 446.415,Z 264.5,A -85,B 0,C 180,E1 -8678.078,E2 -8678.078} C_VEL
LIN {X 0,Y 446.425,Z 264.612,A -85,B 0,C 180,E1 -8679.442,E2 -8679.442} C_VEL
LIN {X 0,Y 447.374,Z 269.777,A -85,B 0,C 180,E1 -8682.493,E2 -8682.493} C_VEL
LIN {X 0,Y 448.284,Z 274.484,A -85,B 0,C 180,E1 -8685.13,E2 -8685.13} C_VEL
LIN {X 0,Y 449.049,Z 279.332,A -85,B 0,C 180,E1 -8687.702,E2 -8687.702} C_VEL
LIN {X 0,Y 448.898,Z 284.225,A -85,B 0,C 180,E1 -8690.098,E2 -8690.098} C_VEL
LIN {X 0,Y 448.413,Z 291.431,A -85,B 0,C 180,E1 -8693.446,E2 -8693.446} C_VEL
LIN {X 0,Y 447.849,Z 298.727,A -85,B 0,C 180,E1 -8696.684,E2 -8696.684} C_VEL
LIN {X 0,Y 447.431,Z 306.081,A -85,B 0,C 180,E1 -8699.825,E2 -8699.825} C_VEL
LIN {X 0,Y 447.037,Z 313.502,A -85,B 0,C 180,E1 -8702.876,E2 -8702.876} C_VEL
LIN {X 0,Y 446.608,Z 322.237,A -85,B 0,C 180,E1 -8706.348,E2 -8706.348} C_VEL
LIN {X 0,Y 446.54,Z 324.047,A -85,B 0,C 180,E1 -8707.064,E2 -8707.064} C_VEL
LIN {X 0,Y 450.952,Z 341.414,A -85,B 0,C 180,E1 -8707.722,E2 -8707.722} C_VEL
LIN {X 0,Y 453.708,Z 354.396,A -85,B 0,C 180,E1 -8708.316,E2 -8708.316} C_VEL
LIN {X 0,Y 452.961,Z 369.543,A -85,B 0,C 180,E1 -8708.992,E2 -8708.992} C_VEL
LIN {X 0,Y 451.859,Z 384.751,A -85,B 0,C 180,E1 -8709.872,E2 -8709.872} C_VEL
LIN {X 0,Y 450.858,Z 398.687,A -85,B 0,C 180,E1 -8710.892,E2 -8710.892} C_VEL
LIN {X 0,Y 449.825,Z 411.658,A -85,B 0,C 180,E1 -8712.05,E2 -8712.05} C_VEL
LIN {X 0,Y 448.841,Z 424.134,A -85,B 0,C 180,E1 -8713.396,E2 -8713.396} C_VEL
LIN {X 0,Y 447.983,Z 434.768,A -85,B 0,C 180,E1 -8714.765,E2 -8714.765} C_VEL
LIN {X 0,Y 447.135,Z 445.164,A -85,B 0,C 180,E1 -8716.363,E2 -8716.363} C_VEL
LIN {X 0,Y 446.549,Z 453.865,A -85,B 0,C 180,E1 -8717.971,E2 -8717.971} C_VEL
LIN {X 0,Y 446.074,Z 461.039,A -85,B 0,C 180,E1 -8719.561,E2 -8719.561} C_VEL
LIN {X 0,Y 445.757,Z 467.728,A -85,B 0,C 180,E1 -8721.386,E2 -8721.386} C_VEL
LIN {X 0,Y 445.535,Z 472.959,A -85,B 0,C 180,E1 -8723.206,E2 -8723.206} C_VEL
LIN {X 0,Y 445.461,Z 475.968,A -85,B 0,C 180,E1 -8724.568,E2 -8724.568} C_VEL
LIN {X 0,Y 445.339,Z 478.922,A -85,B 0,C 180,E1 -8726.381,E2 -8726.381} C_VEL
LIN {X 0,Y 445.348,Z 480.684,A -85,B 0,C 180,E1 -8728.191,E2 -8728.191} C_VEL
LIN {X 0,Y 445.289,Z 481.273,A -85,B 0,C 180,E1 -8730,E2 -8730} C_VEL
LIN {X 0,Y 445.348,Z 480.674,A -85,B 0,C 180,E1 -8731.809,E2 -8731.809} C_VEL
LIN {X 0,Y 445.339,Z 478.897,A -85,B 0,C 180,E1 -8733.619,E2 -8733.619} C_VEL
LIN {X 0,Y 445.471,Z 475.928,A -85,B 0,C 180,E1 -8735.432,E2 -8735.432} C_VEL
LIN {X 0,Y 445.587,Z 471.682,A -85,B 0,C 180,E1 -8737.249,E2 -8737.249} C_VEL
LIN {X 0,Y 445.801,Z 466.053,A -85,B 0,C 180,E1 -8739.07,E2 -8739.07} C_VEL
LIN {X 0,Y 446.228,Z 458.9,A -85,B 0,C 180,E1 -8740.894,E2 -8740.894} C_VEL
LIN {X 0,Y 446.69,Z 450.773,A -85,B 0,C 180,E1 -8742.579,E2 -8742.579} C_VEL
LIN {X 0,Y 447.349,Z 441.995,A -85,B 0,C 180,E1 -8744.094,E2 -8744.094} C_VEL
LIN {X 0,Y 448.181,Z 430.883,A -85,B 0,C 180,E1 -8745.694,E2 -8745.694} C_VEL
LIN {X 0,Y 449.149,Z 418.444,A -85,B 0,C 180,E1 -8747.178,E2 -8747.178} C_VEL
LIN {X 0,Y 450.187,Z 405.782,A -85,B 0,C 180,E1 -8748.429,E2 -8748.429} C_VEL
LIN {X 0,Y 451.243,Z 391.845,A -85,B 0,C 180,E1 -8749.564,E2 -8749.564} C_VEL
LIN {X 0,Y 452.202,Z 378.255,A -85,B 0,C 180,E1 -8750.468,E2 -8750.468} C_VEL
LIN {X 0,Y 453.112,Z 362.767,A -85,B 0,C 180,E1 -8751.288,E2 -8751.288} C_VEL
LIN {X 0,Y 453.501,Z 353.411,A -85,B 0,C 180,E1 -8751.69,E2 -8751.69} C_VEL
LIN {X 0,Y 449.943,Z 337.485,A -85,B 0,C 180,E1 -8752.424,E2 -8752.424} C_VEL
LIN {X 0,Y 446.397,Z 322.34,A -85,B 0,C 180,E1 -8752.995,E2 -8752.995} C_VEL
LIN {X 0,Y 446.742,Z 313.61,A -85,B 0,C 180,E1 -8756.272,E2 -8756.272} C_VEL
LIN {X 0,Y 447.13,Z 304.96,A -85,B 0,C 180,E1 -8759.671,E2 -8759.671} C_VEL
LIN {X 0,Y 447.47,Z 297.529,A -85,B 0,C 180,E1 -8762.811,E2 -8762.811} C_VEL
LIN {X 0,Y 447.973,Z 290.593,A -85,B 0,C 180,E1 -8766.038,E2 -8766.038} C_VEL
LIN {X 0,Y 448.454,Z 285.387,A -85,B 0,C 180,E1 -8768.819,E2 -8768.819} C_VEL
LIN {X 0,Y 448.912,Z 281.522,A -85,B 0,C 180,E1 -8771.282,E2 -8771.282} C_VEL
LIN {X 0,Y 448.999,Z 279.777,A -85,B 0,C 180,E1 -8772.636,E2 -8772.636} C_VEL
LIN {X 0,Y 448.686,Z 277.328,A -85,B 0,C 180,E1 -8775.182,E2 -8775.182} C_VEL
LIN {X 0,Y 448.246,Z 275.922,A -85,B 0,C 180,E1 -8777.609,E2 -8777.609} C_VEL
LIN {X 0,Y 447.653,Z 275.315,A -85,B 0,C 180,E1 -8780.29,E2 -8780.29} C_VEL
LIN {X 0,Y 447.213,Z 275.516,A -85,B 0,C 180,E1 -8783.332,E2 -8783.332} C_VEL
LIN {X 0,Y 446.809,Z 276.493,A -85,B 0,C 180,E1 -8786.597,E2 -8786.597} C_VEL
LIN {X 0,Y 446.55,Z 278.034,A -85,B 0,C 180,E1 -8789.954,E2 -8789.954} C_VEL
LIN {X 0,Y 446.363,Z 279.672,A -85,B 0,C 180,E1 -8792.832,E2 -8792.832} C_VEL
LIN {X 0,Y 446.309,Z 280.093,A -85,B 0,C 180,E1 -8793.51,E2 -8793.51} C_VEL
LIN {X 0,Y 448.358,Z 285.403,A -85,B 0,C 180,E1 -8793.8,E2 -8793.8} C_VEL
LIN {X 0,Y 452.502,Z 297.172,A -85,B 0,C 180,E1 -8794.454,E2 -8794.454} C_VEL
LIN {X 0,Y 453.34,Z 300.518,A -85,B 0,C 180,E1 -8794.635,E2 -8794.635} C_VEL
LIN {X 0,Y 452.642,Z 316.14,A -85,B 0,C 180,E1 -8795.337,E2 -8795.337} C_VEL
LIN {X 0,Y 451.824,Z 330.196,A -85,B 0,C 180,E1 -8796.145,E2 -8796.145} C_VEL
LIN {X 0,Y 450.943,Z 344.687,A -85,B 0,C 180,E1 -8797.19,E2 -8797.19} C_VEL
LIN {X 0,Y 450.135,Z 356.707,A -85,B 0,C 180,E1 -8798.235,E2 -8798.235} C_VEL
LIN {X 0,Y 449.288,Z 367.961,A -85,B 0,C 180,E1 -8799.393,E2 -8799.393} C_VEL
LIN {X 0,Y 448.479,Z 379.278,A -85,B 0,C 180,E1 -8800.787,E2 -8800.787} C_VEL
LIN {X 0,Y 447.75,Z 388.744,A -85,B 0,C 180,E1 -8802.177,E2 -8802.177} C_VEL
LIN {X 0,Y 447.113,Z 398.006,A -85,B 0,C 180,E1 -8803.799,E2 -8803.799} C_VEL
LIN {X 0,Y 446.587,Z 405.597,A -85,B 0,C 180,E1 -8805.417,E2 -8805.417} C_VEL
LIN {X 0,Y 446.175,Z 412.593,A -85,B 0,C 180,E1 -8807.26,E2 -8807.26} C_VEL
LIN {X 0,Y 445.883,Z 417.997,A -85,B 0,C 180,E1 -8809.097,E2 -8809.097} C_VEL
LIN {X 0,Y 445.649,Z 421.979,A -85,B 0,C 180,E1 -8810.927,E2 -8810.927} C_VEL
LIN {X 0,Y 445.566,Z 424.649,A -85,B 0,C 180,E1 -8812.751,E2 -8812.751} C_VEL
LIN {X 0,Y 445.526,Z 426.092,A -85,B 0,C 180,E1 -8814.569,E2 -8814.569} C_VEL
LIN {X 0,Y 445.548,Z 426.342,A -85,B 0,C 180,E1 -8816.383,E2 -8816.383} C_VEL
LIN {X 0,Y 445.517,Z 425.424,A -85,B 0,C 180,E1 -8818.192,E2 -8818.192} C_VEL
LIN {X 0,Y 445.415,Z 423.333,A -85,B 0,C 180,E1 -8820,E2 -8820} C_VEL
LIN {X 0,Y 445.563,Z 419.975,A -85,B 0,C 180,E1 -8821.808,E2 -8821.808} C_VEL
LIN {X 0,Y 445.967,Z 415.311,A -85,B 0,C 180,E1 -8823.614,E2 -8823.614} C_VEL
LIN {X 0,Y 446.235,Z 409.274,A -85,B 0,C 180,E1 -8825.423,E2 -8825.423} C_VEL
LIN {X 0,Y 446.507,Z 402.481,A -85,B 0,C 180,E1 -8827.057,E2 -8827.057} C_VEL
LIN {X 0,Y 447.05,Z 394.779,A -85,B 0,C 180,E1 -8828.589,E2 -8828.589} C_VEL
LIN {X 0,Y 447.723,Z 385.266,A -85,B 0,C 180,E1 -8830.172,E2 -8830.172} C_VEL
LIN {X 0,Y 448.391,Z 375.594,A -85,B 0,C 180,E1 -8831.528,E2 -8831.528} C_VEL
LIN {X 0,Y 449.257,Z 364.124,A -85,B 0,C 180,E1 -8832.881,E2 -8832.881} C_VEL
LIN {X 0,Y 450.135,Z 351.558,A -85,B 0,C 180,E1 -8834.12,E2 -8834.12} C_VEL
LIN {X 0,Y 450.892,Z 339.261,A -85,B 0,C 180,E1 -8835.137,E2 -8835.137} C_VEL
LIN {X 0,Y 451.744,Z 326.15,A -85,B 0,C 180,E1 -8836.031,E2 -8836.031} C_VEL
LIN {X 0,Y 452.464,Z 311.911,A -85,B 0,C 180,E1 -8836.814,E2 -8836.814} C_VEL
LIN {X 0,Y 452.785,Z 298.754,A -85,B 0,C 180,E1 -8837.39,E2 -8837.39} C_VEL
LIN {X 0,Y 448.288,Z 283.204,A -85,B 0,C 180,E1 -8838.118,E2 -8838.118} C_VEL
LIN {X 0,Y 445.689,Z 274.405,A -85,B 0,C 180,E1 -8838.472,E2 -8838.472} C_VEL
LIN {X 0,Y 445.692,Z 271.421,A -85,B 0,C 180,E1 -8841.509,E2 -8841.509} C_VEL
LIN {X 0,Y 445.756,Z 268.816,A -85,B 0,C 180,E1 -8844.201,E2 -8844.201} C_VEL
LIN {X 0,Y 445.76,Z 265.938,A -85,B 0,C 180,E1 -8847.208,E2 -8847.208} C_VEL
LIN {X 0,Y 445.792,Z 264.99,A -85,B 0,C 180,E1 -8848.227,E2 -8848.227} C_VEL
LIN {X 0,Y 445.945,Z 264.564,A -85,B 0,C 180,E1 -8849.912,E2 -8849.912} C_VEL
LIN {X 0,Y 446.178,Z 264.534,A -85,B 0,C 180,E1 -8852.382,E2 -8852.382} C_VEL
LIN {X 0,Y 446.386,Z 264.507,A -85,B 0,C 180,E1 -8855.045,E2 -8855.045} C_VEL
LIN {X 0,Y 446.415,Z 264.502,A -85,B 0,C 180,E1 -8858.079,E2 -8858.079} C_VEL
LIN {X 0,Y 446.426,Z 264.502,A -85,B 0,C 180,E1 -8860.917,E2 -8860.917} C_VEL
LIN {X 0,Y 446.401,Z 264.502,A -85,B 0,C 180,E1 -8863.846,E2 -8863.846} C_VEL
LIN {X 0,Y 446.402,Z 264.506,A -85,B 0,C 180,E1 -8866.403,E2 -8866.403} C_VEL
LIN {X 0,Y 446.431,Z 264.504,A -85,B 0,C 180,E1 -8869.082,E2 -8869.082} C_VEL
LIN {X 0,Y 446.412,Z 264.503,A -85,B 0,C 180,E1 -8872.121,E2 -8872.121} C_VEL
LIN {X 0,Y 446.426,Z 264.501,A -85,B 0,C 180,E1 -8875.476,E2 -8875.476} C_VEL
LIN {X 0,Y 446.419,Z 264.504,A -85,B 0,C 180,E1 -8878.7,E2 -8878.7} C_VEL
LIN {X 0,Y 446.488,Z 264.494,A -85,B 0,C 180,E1 -8881.821,E2 -8881.821} C_VEL
LIN {X 0,Y 446.44,Z 264.5,A -85,B 0,C 180,E1 -8884.846,E2 -8884.846} C_VEL
LIN {X 0,Y 446.452,Z 264.499,A -85,B 0,C 180,E1 -8888.245,E2 -8888.245} C_VEL
LIN {X 0,Y 446.454,Z 264.496,A -85,B 0,C 180,E1 -8891.649,E2 -8891.649} C_VEL
LIN {X 0,Y 446.511,Z 264.492,A -85,B 0,C 180,E1 -8894.48,E2 -8894.48} C_VEL
LIN {X 0,Y 446.521,Z 264.493,A -85,B 0,C 180,E1 -8898.193,E2 -8898.193} C_VEL
LIN {X 0,Y 446.539,Z 264.487,A -85,B 0,C 180,E1 -8901.18,E2 -8901.18} C_VEL
LIN {X 0,Y 445.901,Z 264.568,A -85,B 0,C 180,E1 -8901.933,E2 -8901.933} C_VEL
LIN {X 0,Y 443.1,Z 264.915,A -85,B 0,C 180,E1 -8903.157,E2 -8903.157} C_VEL
LIN {X 0,Y 440.678,Z 265.22,A -85,B 0,C 180,E1 -8904.145,E2 -8904.145} C_VEL
LIN {X 0,Y 439.579,Z 265.352,A -85,B 0,C 180,E1 -8904.907,E2 -8904.907} C_VEL
LIN {X 0,Y 439.459,Z 265.367,A -85,B 0,C 180,E1 -8905.166,E2 -8905.166} C_VEL
LIN {X 0,Y 439.637,Z 265.348,A -85,B 0,C 180,E1 -8908.168,E2 -8908.168} C_VEL
LIN {X 0,Y 439.762,Z 265.333,A -85,B 0,C 180,E1 -8910,E2 -8910} C_VEL
LIN {X 0,Y 439.635,Z 265.346,A -85,B 0,C 180,E1 -8912.749,E2 -8912.749} C_VEL
LIN {X 0,Y 439.596,Z 265.353,A -85,B 0,C 180,E1 -8916.426,E2 -8916.426} C_VEL
LIN {X 0,Y 439.498,Z 265.363,A -85,B 0,C 180,E1 -8919.202,E2 -8919.202} C_VEL
LIN {X 0,Y 439.469,Z 265.368,A -85,B 0,C 180,E1 -8922.938,E2 -8922.938} C_VEL
LIN {X 0,Y 439.45,Z 265.369,A -85,B 0,C 180,E1 -8926.348,E2 -8926.348} C_VEL
LIN {X 0,Y 439.406,Z 265.377,A -85,B 0,C 180,E1 -8929.626,E2 -8929.626} C_VEL
LIN {X 0,Y 439.369,Z 265.378,A -85,B 0,C 180,E1 -8932.575,E2 -8932.575} C_VEL
LIN {X 0,Y 439.409,Z 265.376,A -85,B 0,C 180,E1 -8935.585,E2 -8935.585} C_VEL
LIN {X 0,Y 439.42,Z 265.373,A -85,B 0,C 180,E1 -8938.674,E2 -8938.674} C_VEL
LIN {X 0,Y 439.373,Z 265.38,A -85,B 0,C 180,E1 -8942.03,E2 -8942.03} C_VEL
LIN {X 0,Y 439.397,Z 265.38,A -85,B 0,C 180,E1 -8945.34,E2 -8945.34} C_VEL
LIN {X 0,Y 439.366,Z 265.382,A -85,B 0,C 180,E1 -8948.597,E2 -8948.597} C_VEL
LIN {X 0,Y 439.367,Z 265.383,A -85,B 0,C 180,E1 -8951.253,E2 -8951.253} C_VEL
LIN {X 0,Y 439.401,Z 265.379,A -85,B 0,C 180,E1 -8954.73,E2 -8954.73} C_VEL
LIN {X 0,Y 439.4,Z 265.376,A -85,B 0,C 180,E1 -8957.796,E2 -8957.796} C_VEL
LIN {X 0,Y 439.434,Z 265.371,A -85,B 0,C 180,E1 -8960.228,E2 -8960.228} C_VEL
LIN {X 0,Y 439.377,Z 265.379,A -85,B 0,C 180,E1 -8963.713,E2 -8963.713} C_VEL
LIN {X 0,Y 439.376,Z 265.38,A -85,B 0,C 180,E1 -8967.054,E2 -8967.054} C_VEL
LIN {X 0,Y 439.387,Z 265.379,A -85,B 0,C 180,E1 -8970.274,E2 -8970.274} C_VEL
LIN {X 0,Y 439.423,Z 265.371,A -85,B 0,C 180,E1 -8973.396,E2 -8973.396} C_VEL
LIN {X 0,Y 439.388,Z 265.379,A -85,B 0,C 180,E1 -8976.429,E2 -8976.429} C_VEL
LIN {X 0,Y 439.392,Z 265.376,A -85,B 0,C 180,E1 -8979.397,E2 -8979.397} C_VEL
LIN {X 0,Y 439.429,Z 265.375,A -85,B 0,C 180,E1 -8982.309,E2 -8982.309} C_VEL
LIN {X 0,Y 439.45,Z 265.37,A -85,B 0,C 180,E1 -8985.174,E2 -8985.174} C_VEL
LIN {X 0,Y 439.489,Z 265.367,A -85,B 0,C 180,E1 -8988.001,E2 -8988.001} C_VEL
LIN {X 0,Y 439.508,Z 265.364,A -85,B 0,C 180,E1 -8991.725,E2 -8991.725} C_VEL
LIN {X 0,Y 439.603,Z 265.351,A -85,B 0,C 180,E1 -8994.495,E2 -8994.495} C_VEL
LIN {X 0,Y 439.639,Z 265.348,A -85,B 0,C 180,E1 -8998.168,E2 -8998.168} C_VEL
LIN {X 0,Y 439.761,Z 265.334,A -85,B 0,C 180,E1 -9000,E2 -9000} C_VEL
LIN {X 0,Y 439.645,Z 265.346,A -85,B 0,C 180,E1 -9002.749,E2 -9002.749} C_VEL
LIN {X 0,Y 439.572,Z 265.355,A -85,B 0,C 180,E1 -9006.426,E2 -9006.426} C_VEL
LIN {X 0,Y 439.495,Z 265.365,A -85,B 0,C 180,E1 -9009.202,E2 -9009.202} C_VEL
LIN {X 0,Y 439.469,Z 265.368,A -85,B 0,C 180,E1 -9012.937,E2 -9012.937} C_VEL
LIN {X 0,Y 439.45,Z 265.37,A -85,B 0,C 180,E1 -9016.348,E2 -9016.348} C_VEL
LIN {X 0,Y 439.406,Z 265.377,A -85,B 0,C 180,E1 -9019.626,E2 -9019.626} C_VEL
LIN {X 0,Y 439.367,Z 265.379,A -85,B 0,C 180,E1 -9022.575,E2 -9022.575} C_VEL
LIN {X 0,Y 439.381,Z 265.38,A -85,B 0,C 180,E1 -9025.586,E2 -9025.586} C_VEL
LIN {X 0,Y 439.393,Z 265.376,A -85,B 0,C 180,E1 -9028.675,E2 -9028.675} C_VEL
LIN {X 0,Y 439.372,Z 265.382,A -85,B 0,C 180,E1 -9032.03,E2 -9032.03} C_VEL
LIN {X 0,Y 439.396,Z 265.378,A -85,B 0,C 180,E1 -9035.34,E2 -9035.34} C_VEL
LIN {X 0,Y 439.386,Z 265.455,A -85,B 0,C 180,E1 -9038.962,E2 -9038.962} C_VEL
LIN {X 0,Y 440.341,Z 270.658,A -85,B 0,C 180,E1 -9042.093,E2 -9042.093} C_VEL
LIN {X 0,Y 441.477,Z 276.737,A -85,B 0,C 180,E1 -9045.536,E2 -9045.536} C_VEL
LIN {X 0,Y 442.105,Z 281.595,A -85,B 0,C 180,E1 -9048.113,E2 -9048.113} C_VEL
LIN {X 0,Y 441.867,Z 286.439,A -85,B 0,C 180,E1 -9050.49,E2 -9050.49} C_VEL
LIN {X 0,Y 441.446,Z 292.499,A -85,B 0,C 180,E1 -9053.343,E2 -9053.343} C_VEL
LIN {X 0,Y 440.858,Z 299.797,A -85,B 0,C 180,E1 -9056.634,E2 -9056.634} C_VEL
LIN {X 0,Y 440.41,Z 307.377,A -85,B 0,C 180,E1 -9059.92,E2 -9059.92} C_VEL
LIN {X 0,Y 439.997,Z 314.555,A -85,B 0,C 180,E1 -9062.92,E2 -9062.92} C_VEL
LIN {X 0,Y 439.528,Z 323.216,A -85,B 0,C 180,E1 -9066.437,E2 -9066.437} C_VEL
LIN {X 0,Y 439.505,Z 323.764,A -85,B 0,C 180,E1 -9066.659,E2 -9066.659} C_VEL
LIN {X 0,Y 444.4,Z 342.856,A -85,B 0,C 180,E1 -9067.424,E2 -9067.424} C_VEL
LIN {X 0,Y 447.03,Z 355.587,A -85,B 0,C 180,E1 -9068.038,E2 -9068.038} C_VEL
LIN {X 0,Y 446.168,Z 370.989,A -85,B 0,C 180,E1 -9068.759,E2 -9068.759} C_VEL
LIN {X 0,Y 445.01,Z 386.058,A -85,B 0,C 180,E1 -9069.669,E2 -9069.669} C_VEL
LIN {X 0,Y 443.972,Z 399.657,A -85,B 0,C 180,E1 -9070.704,E2 -9070.704} C_VEL
LIN {X 0,Y 442.882,Z 412.495,A -85,B 0,C 180,E1 -9071.891,E2 -9071.891} C_VEL
LIN {X 0,Y 441.965,Z 423.74,A -85,B 0,C 180,E1 -9073.135,E2 -9073.135} C_VEL
LIN {X 0,Y 441.023,Z 434.33,A -85,B 0,C 180,E1 -9074.519,E2 -9074.519} C_VEL
LIN {X 0,Y 440.139,Z 444.735,A -85,B 0,C 180,E1 -9076.142,E2 -9076.142} C_VEL
LIN {X 0,Y 439.56,Z 452.969,A -85,B 0,C 180,E1 -9077.678,E2 -9077.678} C_VEL
LIN {X 0,Y 439.205,Z 458.684,A -85,B 0,C 180,E1 -9078.929,E2 -9078.929} C_VEL
LIN {X 0,Y 438.732,Z 465.768,A -85,B 0,C 180,E1 -9080.782,E2 -9080.782} C_VEL
LIN {X 0,Y 438.507,Z 471.352,A -85,B 0,C 180,E1 -9082.633,E2 -9082.633} C_VEL
LIN {X 0,Y 438.362,Z 475.575,A -85,B 0,C 180,E1 -9084.48,E2 -9084.48} C_VEL
LIN {X 0,Y 438.245,Z 478.53,A -85,B 0,C 180,E1 -9086.322,E2 -9086.322} C_VEL
LIN {X 0,Y 438.271,Z 480.289,A -85,B 0,C 180,E1 -9088.162,E2 -9088.162} C_VEL
LIN {X 0,Y 438.203,Z 480.872,A -85,B 0,C 180,E1 -9090,E2 -9090} C_VEL
LIN {X 0,Y 438.271,Z 480.263,A -85,B 0,C 180,E1 -9091.838,E2 -9091.838} C_VEL
LIN {X 0,Y 438.335,Z 479.523,A -85,B 0,C 180,E1 -9092.757,E2 -9092.757} C_VEL
LIN {X 0,Y 438.308,Z 477.133,A -85,B 0,C 180,E1 -9094.598,E2 -9094.598} C_VEL
LIN {X 0,Y 438.445,Z 473.514,A -85,B 0,C 180,E1 -9096.442,E2 -9096.442} C_VEL
LIN {X 0,Y 438.605,Z 468.564,A -85,B 0,C 180,E1 -9098.292,E2 -9098.292} C_VEL
LIN {X 0,Y 438.888,Z 462.158,A -85,B 0,C 180,E1 -9100.145,E2 -9100.145} C_VEL
LIN {X 0,Y 439.388,Z 455.239,A -85,B 0,C 180,E1 -9101.767,E2 -9101.767} C_VEL
LIN {X 0,Y 439.911,Z 446.895,A -85,B 0,C 180,E1 -9103.394,E2 -9103.394} C_VEL
LIN {X 0,Y 440.716,Z 436.873,A -85,B 0,C 180,E1 -9105.019,E2 -9105.019} C_VEL
LIN {X 0,Y 441.537,Z 426.64,A -85,B 0,C 180,E1 -9106.411,E2 -9106.411} C_VEL
LIN {X 0,Y 442.547,Z 414.733,A -85,B 0,C 180,E1 -9107.777,E2 -9107.777} C_VEL
LIN {X 0,Y 443.556,Z 402.468,A -85,B 0,C 180,E1 -9108.955,E2 -9108.955} C_VEL
LIN {X 0,Y 444.581,Z 389.543,A -85,B 0,C 180,E1 -9109.99,E2 -9109.99} C_VEL
LIN {X 0,Y 445.632,Z 375.607,A -85,B 0,C 180,E1 -9110.905,E2 -9110.905} C_VEL
LIN {X 0,Y 446.586,Z 360.277,A -85,B 0,C 180,E1 -9111.706,E2 -9111.706} C_VEL
LIN {X 0,Y 446.727,Z 354.413,A -85,B 0,C 180,E1 -9111.969,E2 -9111.969} C_VEL
LIN {X 0,Y 443.524,Z 339.601,A -85,B 0,C 180,E1 -9112.699,E2 -9112.699} C_VEL
LIN {X 0,Y 439.355,Z 321.655,A -85,B 0,C 180,E1 -9113.441,E2 -9113.441} C_VEL
LIN {X 0,Y 439.705,Z 313.503,A -85,B 0,C 180,E1 -9116.586,E2 -9116.586} C_VEL
LIN {X 0,Y 440.097,Z 305.854,A -85,B 0,C 180,E1 -9119.673,E2 -9119.673} C_VEL
LIN {X 0,Y 440.448,Z 298.495,A -85,B 0,C 180,E1 -9122.856,E2 -9122.856} C_VEL
LIN {X 0,Y 440.993,Z 291.646,A -85,B 0,C 180,E1 -9126.133,E2 -9126.133} C_VEL
LIN {X 0,Y 441.47,Z 286.896,A -85,B 0,C 180,E1 -9128.734,E2 -9128.734} C_VEL
LIN {X 0,Y 441.84,Z 283.795,A -85,B 0,C 180,E1 -9130.705,E2 -9130.705} C_VEL
LIN {X 0,Y 442.005,Z 280.863,A -85,B 0,C 180,E1 -9132.995,E2 -9132.995} C_VEL
LIN {X 0,Y 441.676,Z 278.564,A -85,B 0,C 180,E1 -9135.563,E2 -9135.563} C_VEL
LIN {X 0,Y 441.21,Z 277.273,A -85,B 0,C 180,E1 -9138.009,E2 -9138.009} C_VEL
LIN {X 0,Y 440.699,Z 276.758,A -85,B 0,C 180,E1 -9140.365,E2 -9140.365} C_VEL
LIN {X 0,Y 440.299,Z 276.822,A -85,B 0,C 180,E1 -9142.949,E2 -9142.949} C_VEL
LIN {X 0,Y 439.89,Z 277.616,A -85,B 0,C 180,E1 -9146.181,E2 -9146.181} C_VEL
LIN {X 0,Y 439.599,Z 278.872,A -85,B 0,C 180,E1 -9149.23,E2 -9149.23} C_VEL
LIN {X 0,Y 439.397,Z 280.524,A -85,B 0,C 180,E1 -9152.365,E2 -9152.365} C_VEL
LIN {X 0,Y 439.355,Z 281.149,A -85,B 0,C 180,E1 -9153.084,E2 -9153.084} C_VEL
LIN {X 0,Y 444.956,Z 295.616,A -85,B 0,C 180,E1 -9153.937,E2 -9153.937} C_VEL
LIN {X 0,Y 446.804,Z 302.052,A -85,B 0,C 180,E1 -9154.312,E2 -9154.312} C_VEL
LIN {X 0,Y 446.075,Z 317.03,A -85,B 0,C 180,E1 -9155.012,E2 -9155.012} C_VEL
LIN {X 0,Y 445.143,Z 331.657,A -85,B 0,C 180,E1 -9155.882,E2 -9155.882} C_VEL
LIN {X 0,Y 444.221,Z 346.024,A -85,B 0,C 180,E1 -9156.948,E2 -9156.948} C_VEL
LIN {X 0,Y 443.377,Z 357.889,A -85,B 0,C 180,E1 -9158.008,E2 -9158.008} C_VEL
LIN {X 0,Y 442.398,Z 369.987,A -85,B 0,C 180,E1 -9159.301,E2 -9159.301} C_VEL
LIN {X 0,Y 441.567,Z 381.054,A -85,B 0,C 180,E1 -9160.716,E2 -9160.716} C_VEL
LIN {X 0,Y 440.777,Z 390.381,A -85,B 0,C 180,E1 -9162.126,E2 -9162.126} C_VEL
LIN {X 0,Y 440.117,Z 399.57,A -85,B 0,C 180,E1 -9163.807,E2 -9163.807} C_VEL
LIN {X 0,Y 439.481,Z 407.783,A -85,B 0,C 180,E1 -9165.649,E2 -9165.649} C_VEL
LIN {X 0,Y 439.109,Z 414.367,A -85,B 0,C 180,E1 -9167.507,E2 -9167.507} C_VEL
LIN {X 0,Y 438.78,Z 419.497,A -85,B 0,C 180,E1 -9169.386,E2 -9169.386} C_VEL
LIN {X 0,Y 438.598,Z 422.384,A -85,B 0,C 180,E1 -9170.78,E2 -9170.78} C_VEL
LIN {X 0,Y 438.517,Z 425.081,A -85,B 0,C 180,E1 -9172.634,E2 -9172.634} C_VEL
LIN {X 0,Y 438.469,Z 426.555,A -85,B 0,C 180,E1 -9174.481,E2 -9174.481} C_VEL
LIN {X 0,Y 438.484,Z 426.832,A -85,B 0,C 180,E1 -9176.324,E2 -9176.324} C_VEL
LIN {X 0,Y 438.46,Z 425.928,A -85,B 0,C 180,E1 -9178.163,E2 -9178.163} C_VEL
LIN {X 0,Y 438.352,Z 423.84,A -85,B 0,C 180,E1 -9180,E2 -9180} C_VEL
LIN {X 0,Y 438.508,Z 420.479,A -85,B 0,C 180,E1 -9181.837,E2 -9181.837} C_VEL
LIN {X 0,Y 438.912,Z 415.815,A -85,B 0,C 180,E1 -9183.672,E2 -9183.672} C_VEL
LIN {X 0,Y 439.206,Z 409.774,A -85,B 0,C 180,E1 -9185.51,E2 -9185.51} C_VEL
LIN {X 0,Y 439.478,Z 403.208,A -85,B 0,C 180,E1 -9187.12,E2 -9187.12} C_VEL
LIN {X 0,Y 440.065,Z 395.278,A -85,B 0,C 180,E1 -9188.727,E2 -9188.727} C_VEL
LIN {X 0,Y 440.772,Z 385.759,A -85,B 0,C 180,E1 -9190.334,E2 -9190.334} C_VEL
LIN {X 0,Y 441.468,Z 376.085,A -85,B 0,C 180,E1 -9191.711,E2 -9191.711} C_VEL
LIN {X 0,Y 442.376,Z 364.618,A -85,B 0,C 180,E1 -9193.085,E2 -9193.085} C_VEL
LIN {X 0,Y 443.282,Z 352.065,A -85,B 0,C 180,E1 -9194.343,E2 -9194.343} C_VEL
LIN {X 0,Y 444.17,Z 338.432,A -85,B 0,C 180,E1 -9195.475,E2 -9195.475} C_VEL
LIN {X 0,Y 445.055,Z 324.814,A -85,B 0,C 180,E1 -9196.396,E2 -9196.396} C_VEL
LIN {X 0,Y 445.779,Z 311.465,A -85,B 0,C 180,E1 -9197.128,E2 -9197.128} C_VEL
LIN {X 0,Y 446.038,Z 300.151,A -85,B 0,C 180,E1 -9197.635,E2 -9197.635} C_VEL
LIN {X 0,Y 441.59,Z 284.719,A -85,B 0,C 180,E1 -9198.388,E2 -9198.388} C_VEL
LIN {X 0,Y 438.611,Z 274.739,A -85,B 0,C 180,E1 -9198.801,E2 -9198.801} C_VEL
LIN {X 0,Y 438.639,Z 271.938,A -85,B 0,C 180,E1 -9201.674,E2 -9201.674} C_VEL
LIN {X 0,Y 438.712,Z 269.112,A -85,B 0,C 180,E1 -9204.615,E2 -9204.615} C_VEL
LIN {X 0,Y 438.712,Z 266.225,A -85,B 0,C 180,E1 -9207.683,E2 -9207.683} C_VEL
LIN {X 0,Y 438.759,Z 265.459,A -85,B 0,C 180,E1 -9208.721,E2 -9208.721} C_VEL
LIN {X 0,Y 439.118,Z 265.414,A -85,B 0,C 180,E1 -9211.977,E2 -9211.977} C_VEL
LIN {X 0,Y 439.364,Z 265.382,A -85,B 0,C 180,E1 -9215.16,E2 -9215.16} C_VEL
LIN {X 0,Y 439.373,Z 265.381,A -85,B 0,C 180,E1 -9218.596,E2 -9218.596} C_VEL
LIN {X 0,Y 439.385,Z 265.38,A -85,B 0,C 180,E1 -9221.256,E2 -9221.256} C_VEL
LIN {X 0,Y 439.402,Z 265.379,A -85,B 0,C 180,E1 -9224.73,E2 -9224.73} C_VEL
LIN {X 0,Y 439.399,Z 265.377,A -85,B 0,C 180,E1 -9227.796,E2 -9227.796} C_VEL
LIN {X 0,Y 439.414,Z 265.374,A -85,B 0,C 180,E1 -9230.226,E2 -9230.226} C_VEL
LIN {X 0,Y 439.376,Z 265.379,A -85,B 0,C 180,E1 -9233.713,E2 -9233.713} C_VEL
LIN {X 0,Y 439.375,Z 265.38,A -85,B 0,C 180,E1 -9237.054,E2 -9237.054} C_VEL
LIN {X 0,Y 439.386,Z 265.381,A -85,B 0,C 180,E1 -9240.274,E2 -9240.274} C_VEL
LIN {X 0,Y 439.422,Z 265.372,A -85,B 0,C 180,E1 -9243.396,E2 -9243.396} C_VEL
LIN {X 0,Y 439.385,Z 265.38,A -85,B 0,C 180,E1 -9246.429,E2 -9246.429} C_VEL
LIN {X 0,Y 439.391,Z 265.377,A -85,B 0,C 180,E1 -9249.397,E2 -9249.397} C_VEL
LIN {X 0,Y 439.428,Z 265.376,A -85,B 0,C 180,E1 -9252.309,E2 -9252.309} C_VEL
LIN {X 0,Y 439.45,Z 265.37,A -85,B 0,C 180,E1 -9255.174,E2 -9255.174} C_VEL
LIN {X 0,Y 439.487,Z 265.367,A -85,B 0,C 180,E1 -9258.001,E2 -9258.001} C_VEL
LIN {X 0,Y 439.536,Z 265.361,A -85,B 0,C 180,E1 -9261.726,E2 -9261.726} C_VEL
LIN {X 0,Y 439.603,Z 265.351,A -85,B 0,C 180,E1 -9264.496,E2 -9264.496} C_VEL
LIN {X 0,Y 439.459,Z 265.367,A -85,B 0,C 180,E1 -9265.166,E2 -9265.166} C_VEL
LIN {X 0,Y 438.715,Z 265.465,A -85,B 0,C 180,E1 -9265.931,E2 -9265.931} C_VEL
LIN {X 0,Y 435.877,Z 265.817,A -85,B 0,C 180,E1 -9267.177,E2 -9267.177} C_VEL
LIN {X 0,Y 433.569,Z 266.104,A -85,B 0,C 180,E1 -9268.182,E2 -9268.182} C_VEL
LIN {X 0,Y 432.639,Z 266.219,A -85,B 0,C 180,E1 -9268.958,E2 -9268.958} C_VEL
LIN {X 0,Y 432.591,Z 266.224,A -85,B 0,C 180,E1 -9269.22,E2 -9269.22} C_VEL
LIN {X 0,Y 432.731,Z 266.209,A -85,B 0,C 180,E1 -9270,E2 -9270} C_VEL
LIN {X 0,Y 432.587,Z 266.224,A -85,B 0,C 180,E1 -9272.794,E2 -9272.794} C_VEL
LIN {X 0,Y 432.589,Z 266.226,A -85,B 0,C 180,E1 -9275.594,E2 -9275.594} C_VEL
LIN {X 0,Y 432.467,Z 266.239,A -85,B 0,C 180,E1 -9278.41,E2 -9278.41} C_VEL
LIN {X 0,Y 432.462,Z 266.242,A -85,B 0,C 180,E1 -9282.197,E2 -9282.197} C_VEL
LIN {X 0,Y 432.433,Z 266.244,A -85,B 0,C 180,E1 -9286.039,E2 -9286.039} C_VEL
LIN {X 0,Y 432.39,Z 266.251,A -85,B 0,C 180,E1 -9289.485,E2 -9289.485} C_VEL
LIN {X 0,Y 432.323,Z 266.257,A -85,B 0,C 180,E1 -9292.964,E2 -9292.964} C_VEL
LIN {X 0,Y 432.368,Z 266.253,A -85,B 0,C 180,E1 -9296.032,E2 -9296.032} C_VEL
LIN {X 0,Y 432.346,Z 266.257,A -85,B 0,C 180,E1 -9299.188,E2 -9299.188} C_VEL
LIN {X 0,Y 432.326,Z 266.258,A -85,B 0,C 180,E1 -9302.443,E2 -9302.443} C_VEL
LIN {X 0,Y 432.347,Z 266.255,A -85,B 0,C 180,E1 -9305.632,E2 -9305.632} C_VEL
LIN {X 0,Y 432.329,Z 266.259,A -85,B 0,C 180,E1 -9308.712,E2 -9308.712} C_VEL
LIN {X 0,Y 432.308,Z 266.259,A -85,B 0,C 180,E1 -9311.801,E2 -9311.801} C_VEL
LIN {X 0,Y 432.337,Z 266.256,A -85,B 0,C 180,E1 -9314.347,E2 -9314.347} C_VEL
LIN {X 0,Y 432.324,Z 266.259,A -85,B 0,C 180,E1 -9317.016,E2 -9317.016} C_VEL
LIN {X 0,Y 432.34,Z 266.253,A -85,B 0,C 180,E1 -9319.82,E2 -9319.82} C_VEL
LIN {X 0,Y 432.311,Z 266.261,A -85,B 0,C 180,E1 -9323.022,E2 -9323.022} C_VEL
LIN {X 0,Y 432.361,Z 266.252,A -85,B 0,C 180,E1 -9325.997,E2 -9325.997} C_VEL
LIN {X 0,Y 432.352,Z 266.255,A -85,B 0,C 180,E1 -9329.49,E2 -9329.49} C_VEL
LIN {X 0,Y 432.39,Z 266.251,A -85,B 0,C 180,E1 -9332.928,E2 -9332.928} C_VEL
LIN {X 0,Y 432.372,Z 266.253,A -85,B 0,C 180,E1 -9336.023,E2 -9336.023} C_VEL
LIN {X 0,Y 432.354,Z 266.254,A -85,B 0,C 180,E1 -9339.046,E2 -9339.046} C_VEL
LIN {X 0,Y 432.377,Z 266.253,A -85,B 0,C 180,E1 -9342.011,E2 -9342.011} C_VEL
LIN {X 0,Y 432.398,Z 266.249,A -85,B 0,C 180,E1 -9344.926,E2 -9344.926} C_VEL
LIN {X 0,Y 432.464,Z 266.24,A -85,B 0,C 180,E1 -9347.803,E2 -9347.803} C_VEL
LIN {X 0,Y 432.468,Z 266.241,A -85,B 0,C 180,E1 -9351.59,E2 -9351.59} C_VEL
LIN {X 0,Y 432.577,Z 266.227,A -85,B 0,C 180,E1 -9354.406,E2 -9354.406} C_VEL
LIN {X 0,Y 432.608,Z 266.224,A -85,B 0,C 180,E1 -9358.138,E2 -9358.138} C_VEL
LIN {X 0,Y 432.73,Z 266.21,A -85,B 0,C 180,E1 -9360,E2 -9360} C_VEL
LIN {X 0,Y 432.596,Z 266.224,A -85,B 0,C 180,E1 -9362.793,E2 -9362.793} C_VEL
LIN {X 0,Y 432.586,Z 266.226,A -85,B 0,C 180,E1 -9365.594,E2 -9365.594} C_VEL
LIN {X 0,Y 432.466,Z 266.239,A -85,B 0,C 180,E1 -9368.41,E2 -9368.41} C_VEL
LIN {X 0,Y 432.463,Z 266.242,A -85,B 0,C 180,E1 -9372.196,E2 -9372.196} C_VEL
LIN {X 0,Y 432.434,Z 266.244,A -85,B 0,C 180,E1 -9376.039,E2 -9376.039} C_VEL
LIN {X 0,Y 432.39,Z 266.251,A -85,B 0,C 180,E1 -9379.485,E2 -9379.485} C_VEL
LIN {X 0,Y 432.321,Z 266.259,A -85,B 0,C 180,E1 -9382.964,E2 -9382.964} C_VEL
LIN {X 0,Y 432.341,Z 266.258,A -85,B 0,C 180,E1 -9385.002,E2 -9385.002} C_VEL
LIN {X 0,Y 432.342,Z 266.254,A -85,B 0,C 180,E1 -9388.126,E2 -9388.126} C_VEL
LIN {X 0,Y 432.322,Z 266.259,A -85,B 0,C 180,E1 -9391.346,E2 -9391.346} C_VEL
LIN {X 0,Y 432.341,Z 266.256,A -85,B 0,C 180,E1 -9394.677,E2 -9394.677} C_VEL
LIN {X 0,Y 432.339,Z 266.254,A -85,B 0,C 180,E1 -9398.438,E2 -9398.438} C_VEL
LIN {X 0,Y 433.327,Z 271.631,A -85,B 0,C 180,E1 -9401.749,E2 -9401.749} C_VEL
LIN {X 0,Y 434.241,Z 276.529,A -85,B 0,C 180,E1 -9404.592,E2 -9404.592} C_VEL
LIN {X 0,Y 435.055,Z 281.41,A -85,B 0,C 180,E1 -9407.275,E2 -9407.275} C_VEL
LIN {X 0,Y 435.067,Z 285.56,A -85,B 0,C 180,E1 -9409.396,E2 -9409.396} C_VEL
LIN {X 0,Y 434.579,Z 291.805,A -85,B 0,C 180,E1 -9412.413,E2 -9412.413} C_VEL
LIN {X 0,Y 434.027,Z 298.834,A -85,B 0,C 180,E1 -9415.671,E2 -9415.671} C_VEL
LIN {X 0,Y 433.493,Z 306.827,A -85,B 0,C 180,E1 -9419.233,E2 -9419.233} C_VEL
LIN {X 0,Y 433.087,Z 313.104,A -85,B 0,C 180,E1 -9421.926,E2 -9421.926} C_VEL
LIN {X 0,Y 432.604,Z 321.616,A -85,B 0,C 180,E1 -9425.473,E2 -9425.473} C_VEL
LIN {X 0,Y 432.486,Z 323.517,A -85,B 0,C 180,E1 -9426.256,E2 -9426.256} C_VEL
LIN {X 0,Y 437.098,Z 341.491,A -85,B 0,C 180,E1 -9426.986,E2 -9426.986} C_VEL
LIN {X 0,Y 440.306,Z 356.203,A -85,B 0,C 180,E1 -9427.725,E2 -9427.725} C_VEL
LIN {X 0,Y 439.449,Z 371.702,A -85,B 0,C 180,E1 -9428.479,E2 -9428.479} C_VEL
LIN {X 0,Y 438.317,Z 385.652,A -85,B 0,C 180,E1 -9429.344,E2 -9429.344} C_VEL
LIN {X 0,Y 437.226,Z 399.231,A -85,B 0,C 180,E1 -9430.394,E2 -9430.394} C_VEL
LIN {X 0,Y 436.115,Z 411.715,A -85,B 0,C 180,E1 -9431.563,E2 -9431.563} C_VEL
LIN {X 0,Y 435.078,Z 423.517,A -85,B 0,C 180,E1 -9432.887,E2 -9432.887} C_VEL
LIN {X 0,Y 434.1,Z 433.895,A -85,B 0,C 180,E1 -9434.265,E2 -9434.265} C_VEL
LIN {X 0,Y 433.169,Z 444.305,A -85,B 0,C 180,E1 -9435.914,E2 -9435.914} C_VEL
LIN {X 0,Y 432.516,Z 452.85,A -85,B 0,C 180,E1 -9437.538,E2 -9437.538} C_VEL
LIN {X 0,Y 432.01,Z 460.214,A -85,B 0,C 180,E1 -9439.217,E2 -9439.217} C_VEL
LIN {X 0,Y 431.587,Z 466.915,A -85,B 0,C 180,E1 -9441.101,E2 -9441.101} C_VEL
LIN {X 0,Y 431.388,Z 472.163,A -85,B 0,C 180,E1 -9442.982,E2 -9442.982} C_VEL
LIN {X 0,Y 431.268,Z 475.183,A -85,B 0,C 180,E1 -9444.389,E2 -9444.389} C_VEL
LIN {X 0,Y 431.153,Z 478.137,A -85,B 0,C 180,E1 -9446.261,E2 -9446.261} C_VEL
LIN {X 0,Y 431.262,Z 479.167,A -85,B 0,C 180,E1 -9447.198,E2 -9447.198} C_VEL
LIN {X 0,Y 431.145,Z 480.331,A -85,B 0,C 180,E1 -9449.066,E2 -9449.066} C_VEL
LIN {X 0,Y 431.145,Z 480.306,A -85,B 0,C 180,E1 -9450.934,E2 -9450.934} C_VEL
LIN {X 0,Y 431.262,Z 479.101,A -85,B 0,C 180,E1 -9452.802,E2 -9452.802} C_VEL
LIN {X 0,Y 431.236,Z 476.701,A -85,B 0,C 180,E1 -9454.674,E2 -9454.674} C_VEL
LIN {X 0,Y 431.373,Z 473.058,A -85,B 0,C 180,E1 -9456.549,E2 -9456.549} C_VEL
LIN {X 0,Y 431.521,Z 468.078,A -85,B 0,C 180,E1 -9458.429,E2 -9458.429} C_VEL
LIN {X 0,Y 431.834,Z 461.641,A -85,B 0,C 180,E1 -9460.313,E2 -9460.313} C_VEL
LIN {X 0,Y 432.352,Z 454.687,A -85,B 0,C 180,E1 -9461.962,E2 -9461.962} C_VEL
LIN {X 0,Y 432.918,Z 446.305,A -85,B 0,C 180,E1 -9463.615,E2 -9463.615} C_VEL
LIN {X 0,Y 433.764,Z 436.247,A -85,B 0,C 180,E1 -9465.265,E2 -9465.265} C_VEL
LIN {X 0,Y 434.639,Z 425.973,A -85,B 0,C 180,E1 -9466.679,E2 -9466.679} C_VEL
LIN {X 0,Y 435.724,Z 413.817,A -85,B 0,C 180,E1 -9468.089,E2 -9468.089} C_VEL
LIN {X 0,Y 436.866,Z 400.447,A -85,B 0,C 180,E1 -9469.378,E2 -9469.378} C_VEL
LIN {X 0,Y 438.093,Z 385.683,A -85,B 0,C 180,E1 -9470.544,E2 -9470.544} C_VEL
LIN {X 0,Y 439.26,Z 371.079,A -85,B 0,C 180,E1 -9471.469,E2 -9471.469} C_VEL
LIN {X 0,Y 440.112,Z 355.914,A -85,B 0,C 180,E1 -9472.233,E2 -9472.233} C_VEL
LIN {X 0,Y 436.38,Z 338.396,A -85,B 0,C 180,E1 -9473.142,E2 -9473.142} C_VEL
LIN {X 0,Y 432.331,Z 320.969,A -85,B 0,C 180,E1 -9473.919,E2 -9473.919} C_VEL
LIN {X 0,Y 432.681,Z 313.066,A -85,B 0,C 180,E1 -9477.052,E2 -9477.052} C_VEL
LIN {X 0,Y 433.051,Z 306.76,A -85,B 0,C 180,E1 -9479.669,E2 -9479.669} C_VEL
LIN {X 0,Y 433.456,Z 299.415,A -85,B 0,C 180,E1 -9482.931,E2 -9482.931} C_VEL
LIN {X 0,Y 433.946,Z 293.297,A -85,B 0,C 180,E1 -9485.926,E2 -9485.926} C_VEL
LIN {X 0,Y 434.568,Z 287.693,A -85,B 0,C 180,E1 -9489.079,E2 -9489.079} C_VEL
LIN {X 0,Y 434.984,Z 284.161,A -85,B 0,C 180,E1 -9491.486,E2 -9491.486} C_VEL
LIN {X 0,Y 435.018,Z 281.976,A -85,B 0,C 180,E1 -9493.364,E2 -9493.364} C_VEL
LIN {X 0,Y 434.676,Z 279.817,A -85,B 0,C 180,E1 -9495.954,E2 -9495.954} C_VEL
LIN {X 0,Y 434.178,Z 278.628,A -85,B 0,C 180,E1 -9498.42,E2 -9498.42} C_VEL
LIN {X 0,Y 433.616,Z 278.149,A -85,B 0,C 180,E1 -9501.076,E2 -9501.076} C_VEL
LIN {X 0,Y 433.32,Z 278.228,A -85,B 0,C 180,E1 -9503.123,E2 -9503.123} C_VEL
LIN {X 0,Y 432.852,Z 279.022,A -85,B 0,C 180,E1 -9506.493,E2 -9506.493} C_VEL
LIN {X 0,Y 432.572,Z 280.339,A -85,B 0,C 180,E1 -9509.758,E2 -9509.758} C_VEL
LIN {X 0,Y 432.372,Z 281.809,A -85,B 0,C 180,E1 -9512.587,E2 -9512.587} C_VEL
LIN {X 0,Y 435.341,Z 289.104,A -85,B 0,C 180,E1 -9513.055,E2 -9513.055} C_VEL
LIN {X 0,Y 439.213,Z 299.649,A -85,B 0,C 180,E1 -9513.732,E2 -9513.732} C_VEL
LIN {X 0,Y 440.271,Z 304.309,A -85,B 0,C 180,E1 -9514.007,E2 -9514.007} C_VEL
LIN {X 0,Y 439.41,Z 320.108,A -85,B 0,C 180,E1 -9514.796,E2 -9514.796} C_VEL
LIN {X 0,Y 438.367,Z 335.17,A -85,B 0,C 180,E1 -9515.744,E2 -9515.744} C_VEL
LIN {X 0,Y 437.366,Z 348.856,A -85,B 0,C 180,E1 -9516.816,E2 -9516.816} C_VEL
LIN {X 0,Y 436.301,Z 362.62,A -85,B 0,C 180,E1 -9518.13,E2 -9518.13} C_VEL
LIN {X 0,Y 435.392,Z 373.9,A -85,B 0,C 180,E1 -9519.428,E2 -9519.428} C_VEL
LIN {X 0,Y 434.5,Z 384.507,A -85,B 0,C 180,E1 -9520.881,E2 -9520.881} C_VEL
LIN {X 0,Y 433.564,Z 394.697,A -85,B 0,C 180,E1 -9522.55,E2 -9522.55} C_VEL
LIN {X 0,Y 432.917,Z 403.074,A -85,B 0,C 180,E1 -9524.222,E2 -9524.222} C_VEL
LIN {X 0,Y 432.418,Z 409.926,A -85,B 0,C 180,E1 -9525.89,E2 -9525.89} C_VEL
LIN {X 0,Y 431.961,Z 416.193,A -85,B 0,C 180,E1 -9527.789,E2 -9527.789} C_VEL
LIN {X 0,Y 431.626,Z 420.956,A -85,B 0,C 180,E1 -9529.682,E2 -9529.682} C_VEL
LIN {X 0,Y 431.479,Z 424.333,A -85,B 0,C 180,E1 -9531.571,E2 -9531.571} C_VEL
LIN {X 0,Y 431.427,Z 426.526,A -85,B 0,C 180,E1 -9533.567,E2 -9533.567} C_VEL
LIN {X 0,Y 431.315,Z 427.33,A -85,B 0,C 180,E1 -9535.327,E2 -9535.327} C_VEL
LIN {X 0,Y 431.386,Z 427.024,A -85,B 0,C 180,E1 -9537.199,E2 -9537.199} C_VEL
LIN {X 0,Y 431.313,Z 425.546,A -85,B 0,C 180,E1 -9539.067,E2 -9539.067} C_VEL
LIN {X 0,Y 431.331,Z 422.824,A -85,B 0,C 180,E1 -9540.934,E2 -9540.934} C_VEL
LIN {X 0,Y 431.636,Z 418.819,A -85,B 0,C 180,E1 -9542.8,E2 -9542.8} C_VEL
LIN {X 0,Y 431.987,Z 413.481,A -85,B 0,C 180,E1 -9544.666,E2 -9544.666} C_VEL
LIN {X 0,Y 432.204,Z 408.536,A -85,B 0,C 180,E1 -9546.067,E2 -9546.067} C_VEL
LIN {X 0,Y 432.685,Z 401.279,A -85,B 0,C 180,E1 -9547.772,E2 -9547.772} C_VEL
LIN {X 0,Y 433.348,Z 391.913,A -85,B 0,C 180,E1 -9549.569,E2 -9549.569} C_VEL
LIN {X 0,Y 434.217,Z 381.602,A -85,B 0,C 180,E1 -9551.2,E2 -9551.2} C_VEL
LIN {X 0,Y 435.016,Z 371.095,A -85,B 0,C 180,E1 -9552.598,E2 -9552.598} C_VEL
LIN {X 0,Y 435.883,Z 359.713,A -85,B 0,C 180,E1 -9553.877,E2 -9553.877} C_VEL
LIN {X 0,Y 436.837,Z 346.272,A -85,B 0,C 180,E1 -9555.136,E2 -9555.136} C_VEL
LIN {X 0,Y 437.83,Z 332.451,A -85,B 0,C 180,E1 -9556.195,E2 -9556.195} C_VEL
LIN {X 0,Y 438.687,Z 317.579,A -85,B 0,C 180,E1 -9557.115,E2 -9557.115} C_VEL
LIN {X 0,Y 439.423,Z 302.487,A -85,B 0,C 180,E1 -9557.841,E2 -9557.841} C_VEL
LIN {X 0,Y 435.566,Z 288.467,A -85,B 0,C 180,E1 -9558.556,E2 -9558.556} C_VEL
LIN {X 0,Y 431.555,Z 275.141,A -85,B 0,C 180,E1 -9559.12,E2 -9559.12} C_VEL
LIN {X 0,Y 431.559,Z 272.338,A -85,B 0,C 180,E1 -9561.997,E2 -9561.997} C_VEL
LIN {X 0,Y 431.65,Z 269.418,A -85,B 0,C 180,E1 -9565.045,E2 -9565.045} C_VEL
LIN {X 0,Y 431.687,Z 266.341,A -85,B 0,C 180,E1 -9568.461,E2 -9568.461} C_VEL
LIN {X 0,Y 431.996,Z 266.303,A -85,B 0,C 180,E1 -9571.373,E2 -9571.373} C_VEL
LIN {X 0,Y 432.281,Z 266.264,A -85,B 0,C 180,E1 -9574.683,E2 -9574.683} C_VEL
LIN {X 0,Y 432.323,Z 266.26,A -85,B 0,C 180,E1 -9577.197,E2 -9577.197} C_VEL
LIN {X 0,Y 432.324,Z 266.26,A -85,B 0,C 180,E1 -9580.561,E2 -9580.561} C_VEL
LIN {X 0,Y 432.317,Z 266.262,A -85,B 0,C 180,E1 -9583.061,E2 -9583.061} C_VEL
LIN {X 0,Y 432.336,Z 266.256,A -85,B 0,C 180,E1 -9585.665,E2 -9585.665} C_VEL
LIN {X 0,Y 432.336,Z 266.257,A -85,B 0,C 180,E1 -9588.398,E2 -9588.398} C_VEL
LIN {X 0,Y 432.339,Z 266.255,A -85,B 0,C 180,E1 -9591.85,E2 -9591.85} C_VEL
LIN {X 0,Y 432.341,Z 266.256,A -85,B 0,C 180,E1 -9595.323,E2 -9595.323} C_VEL
LIN {X 0,Y 432.324,Z 266.26,A -85,B 0,C 180,E1 -9598.654,E2 -9598.654} C_VEL
LIN {X 0,Y 432.383,Z 266.251,A -85,B 0,C 180,E1 -9601.877,E2 -9601.877} C_VEL
LIN {X 0,Y 432.343,Z 266.255,A -85,B 0,C 180,E1 -9604.998,E2 -9604.998} C_VEL
LIN {X 0,Y 432.361,Z 266.255,A -85,B 0,C 180,E1 -9608.046,E2 -9608.046} C_VEL
LIN {X 0,Y 432.387,Z 266.248,A -85,B 0,C 180,E1 -9611.03,E2 -9611.03} C_VEL
LIN {X 0,Y 432.433,Z 266.247,A -85,B 0,C 180,E1 -9613.961,E2 -9613.961} C_VEL
LIN {X 0,Y 432.462,Z 266.24,A -85,B 0,C 180,E1 -9617.803,E2 -9617.803} C_VEL
LIN {X 0,Y 432.486,Z 266.239,A -85,B 0,C 180,E1 -9621.59,E2 -9621.59} C_VEL
LIN {X 0,Y 432.577,Z 266.227,A -85,B 0,C 180,E1 -9624.406,E2 -9624.406} C_VEL
LIN {X 0,Y 432.606,Z 266.224,A -85,B 0,C 180,E1 -9628.138,E2 -9628.138} C_VEL
LIN {X 0,Y 432.591,Z 266.224,A -85,B 0,C 180,E1 -9629.22,E2 -9629.22} C_VEL
LIN {X 0,Y 432.01,Z 266.299,A -85,B 0,C 180,E1 -9629.998,E2 -9629.998} C_VEL
LIN {X 0,Y 429.197,Z 266.646,A -85,B 0,C 180,E1 -9631.261,E2 -9631.261} C_VEL
LIN {X 0,Y 426.707,Z 266.958,A -85,B 0,C 180,E1 -9632.281,E2 -9632.281} C_VEL
LIN {X 0,Y 425.55,Z 267.1,A -85,B 0,C 180,E1 -9633.069,E2 -9633.069} C_VEL
LIN {X 0,Y 425.412,Z 267.117,A -85,B 0,C 180,E1 -9633.336,E2 -9633.336} C_VEL
LIN {X 0,Y 425.545,Z 267.103,A -85,B 0,C 180,E1 -9635.687,E2 -9635.687} C_VEL
LIN {X 0,Y 425.411,Z 267.117,A -85,B 0,C 180,E1 -9638.551,E2 -9638.551} C_VEL
LIN {X 0,Y 425.415,Z 267.119,A -85,B 0,C 180,E1 -9642.402,E2 -9642.402} C_VEL
LIN {X 0,Y 425.391,Z 267.12,A -85,B 0,C 180,E1 -9646.312,E2 -9646.312} C_VEL
LIN {X 0,Y 425.332,Z 267.13,A -85,B 0,C 180,E1 -9649.636,E2 -9649.636} C_VEL
LIN {X 0,Y 425.311,Z 267.135,A -85,B 0,C 180,E1 -9653.365,E2 -9653.365} C_VEL
LIN {X 0,Y 425.351,Z 267.127,A -85,B 0,C 180,E1 -9656.844,E2 -9656.844} C_VEL
LIN {X 0,Y 425.294,Z 267.133,A -85,B 0,C 180,E1 -9659.72,E2 -9659.72} C_VEL
LIN {X 0,Y 425.286,Z 267.136,A -85,B 0,C 180,E1 -9663.048,E2 -9663.048} C_VEL
LIN {X 0,Y 425.284,Z 267.133,A -85,B 0,C 180,E1 -9665.928,E2 -9665.928} C_VEL
LIN {X 0,Y 425.265,Z 267.138,A -85,B 0,C 180,E1 -9669.037,E2 -9669.037} C_VEL
LIN {X 0,Y 425.26,Z 267.138,A -85,B 0,C 180,E1 -9672.655,E2 -9672.655} C_VEL
LIN {X 0,Y 425.288,Z 267.135,A -85,B 0,C 180,E1 -9675.283,E2 -9675.283} C_VEL
LIN {X 0,Y 425.279,Z 267.136,A -85,B 0,C 180,E1 -9678.621,E2 -9678.621} C_VEL
LIN {X 0,Y 425.314,Z 267.132,A -85,B 0,C 180,E1 -9681.103,E2 -9681.103} C_VEL
LIN {X 0,Y 425.302,Z 267.134,A -85,B 0,C 180,E1 -9684.664,E2 -9684.664} C_VEL
LIN {X 0,Y 425.269,Z 267.136,A -85,B 0,C 180,E1 -9688.073,E2 -9688.073} C_VEL
LIN {X 0,Y 425.336,Z 267.128,A -85,B 0,C 180,E1 -9691.368,E2 -9691.368} C_VEL
LIN {X 0,Y 425.289,Z 267.137,A -85,B 0,C 180,E1 -9694.554,E2 -9694.554} C_VEL
LIN {X 0,Y 425.289,Z 267.135,A -85,B 0,C 180,E1 -9696.634,E2 -9696.634} C_VEL
LIN {X 0,Y 425.299,Z 267.132,A -85,B 0,C 180,E1 -9699.694,E2 -9699.694} C_VEL
LIN {X 0,Y 425.344,Z 267.128,A -85,B 0,C 180,E1 -9702.697,E2 -9702.697} C_VEL
LIN {X 0,Y 425.35,Z 267.127,A -85,B 0,C 180,E1 -9705.65,E2 -9705.65} C_VEL
LIN {X 0,Y 425.355,Z 267.126,A -85,B 0,C 180,E1 -9708.564,E2 -9708.564} C_VEL
LIN {X 0,Y 425.413,Z 267.119,A -85,B 0,C 180,E1 -9711.449,E2 -9711.449} C_VEL
LIN {X 0,Y 425.532,Z 267.105,A -85,B 0,C 180,E1 -9714.313,E2 -9714.313} C_VEL
LIN {X 0,Y 425.577,Z 267.1,A -85,B 0,C 180,E1 -9718.107,E2 -9718.107} C_VEL
LIN {X 0,Y 425.699,Z 267.085,A -85,B 0,C 180,E1 -9720,E2 -9720} C_VEL
LIN {X 0,Y 425.55,Z 267.101,A -85,B 0,C 180,E1 -9722.84,E2 -9722.84} C_VEL
LIN {X 0,Y 425.54,Z 267.104,A -85,B 0,C 180,E1 -9725.687,E2 -9725.687} C_VEL
LIN {X 0,Y 425.41,Z 267.118,A -85,B 0,C 180,E1 -9728.55,E2 -9728.55} C_VEL
LIN {X 0,Y 425.416,Z 267.118,A -85,B 0,C 180,E1 -9732.401,E2 -9732.401} C_VEL
LIN {X 0,Y 425.392,Z 267.121,A -85,B 0,C 180,E1 -9736.311,E2 -9736.311} C_VEL
LIN {X 0,Y 425.332,Z 267.131,A -85,B 0,C 180,E1 -9739.635,E2 -9739.635} C_VEL
LIN {X 0,Y 425.308,Z 267.134,A -85,B 0,C 180,E1 -9743.365,E2 -9743.365} C_VEL
LIN {X 0,Y 425.3,Z 267.134,A -85,B 0,C 180,E1 -9746.498,E2 -9746.498} C_VEL
LIN {X 0,Y 425.285,Z 267.135,A -85,B 0,C 180,E1 -9749.72,E2 -9749.72} C_VEL
LIN {X 0,Y 425.284,Z 267.136,A -85,B 0,C 180,E1 -9753.048,E2 -9753.048} C_VEL
LIN {X 0,Y 425.284,Z 267.135,A -85,B 0,C 180,E1 -9755.928,E2 -9755.928} C_VEL
LIN {X 0,Y 425.306,Z 267.148,A -85,B 0,C 180,E1 -9757.991,E2 -9757.991} C_VEL
LIN {X 0,Y 426.224,Z 272.379,A -85,B 0,C 180,E1 -9761.266,E2 -9761.266} C_VEL
LIN {X 0,Y 427.215,Z 277.609,A -85,B 0,C 180,E1 -9764.359,E2 -9764.359} C_VEL
LIN {X 0,Y 428.04,Z 282.416,A -85,B 0,C 180,E1 -9767.048,E2 -9767.048} C_VEL
LIN {X 0,Y 428.125,Z 286.222,A -85,B 0,C 180,E1 -9769.036,E2 -9769.036} C_VEL
LIN {X 0,Y 427.638,Z 292.39,A -85,B 0,C 180,E1 -9772.078,E2 -9772.078} C_VEL
LIN {X 0,Y 427.069,Z 299.353,A -85,B 0,C 180,E1 -9775.368,E2 -9775.368} C_VEL
LIN {X 0,Y 426.504,Z 307.288,A -85,B 0,C 180,E1 -9778.966,E2 -9778.966} C_VEL
LIN {X 0,Y 426.036,Z 314.114,A -85,B 0,C 180,E1 -9781.956,E2 -9781.956} C_VEL
LIN {X 0,Y 425.562,Z 321.919,A -85,B 0,C 180,E1 -9785.272,E2 -9785.272} C_VEL
LIN {X 0,Y 425.493,Z 323.253,A -85,B 0,C 180,E1 -9785.831,E2 -9785.831} C_VEL
LIN {X 0,Y 430.04,Z 340.947,A -85,B 0,C 180,E1 -9786.574,E2 -9786.574} C_VEL
LIN {X 0,Y 433.578,Z 357.051,A -85,B 0,C 180,E1 -9787.411,E2 -9787.411} C_VEL
LIN {X 0,Y 432.729,Z 372.378,A -85,B 0,C 180,E1 -9788.191,E2 -9788.191} C_VEL
LIN {X 0,Y 431.478,Z 386.908,A -85,B 0,C 180,E1 -9789.126,E2 -9789.126} C_VEL
LIN {X 0,Y 430.35,Z 400.169,A -85,B 0,C 180,E1 -9790.192,E2 -9790.192} C_VEL
LIN {X 0,Y 429.071,Z 413.542,A -85,B 0,C 180,E1 -9791.497,E2 -9791.497} C_VEL
LIN {X 0,Y 428.048,Z 424.738,A -85,B 0,C 180,E1 -9792.81,E2 -9792.81} C_VEL
LIN {X 0,Y 427.033,Z 435.086,A -85,B 0,C 180,E1 -9794.243,E2 -9794.243} C_VEL
LIN {X 0,Y 426.07,Z 445.226,A -85,B 0,C 180,E1 -9795.918,E2 -9795.918} C_VEL
LIN {X 0,Y 425.426,Z 453.689,A -85,B 0,C 180,E1 -9797.598,E2 -9797.598} C_VEL
LIN {X 0,Y 424.998,Z 459.802,A -85,B 0,C 180,E1 -9799.037,E2 -9799.037} C_VEL
LIN {X 0,Y 424.524,Z 466.509,A -85,B 0,C 180,E1 -9800.951,E2 -9800.951} C_VEL
LIN {X 0,Y 424.315,Z 471.765,A -85,B 0,C 180,E1 -9802.864,E2 -9802.864} C_VEL
LIN {X 0,Y 424.179,Z 474.789,A -85,B 0,C 180,E1 -9804.295,E2 -9804.295} C_VEL
LIN {X 0,Y 424.066,Z 477.743,A -85,B 0,C 180,E1 -9806.199,E2 -9806.199} C_VEL
LIN {X 0,Y 424.172,Z 478.773,A -85,B 0,C 180,E1 -9807.151,E2 -9807.151} C_VEL
LIN {X 0,Y 424.066,Z 479.934,A -85,B 0,C 180,E1 -9809.05,E2 -9809.05} C_VEL
LIN {X 0,Y 424.066,Z 479.899,A -85,B 0,C 180,E1 -9810.95,E2 -9810.95} C_VEL
LIN {X 0,Y 424.172,Z 478.677,A -85,B 0,C 180,E1 -9812.849,E2 -9812.849} C_VEL
LIN {X 0,Y 424.165,Z 476.259,A -85,B 0,C 180,E1 -9814.752,E2 -9814.752} C_VEL
LIN {X 0,Y 424.295,Z 472.601,A -85,B 0,C 180,E1 -9816.658,E2 -9816.658} C_VEL
LIN {X 0,Y 424.451,Z 467.593,A -85,B 0,C 180,E1 -9818.57,E2 -9818.57} C_VEL
LIN {X 0,Y 424.796,Z 461.125,A -85,B 0,C 180,E1 -9820.486,E2 -9820.486} C_VEL
LIN {X 0,Y 425.333,Z 454.136,A -85,B 0,C 180,E1 -9822.162,E2 -9822.162} C_VEL
LIN {X 0,Y 425.92,Z 445.712,A -85,B 0,C 180,E1 -9823.843,E2 -9823.843} C_VEL
LIN {X 0,Y 426.81,Z 435.615,A -85,B 0,C 180,E1 -9825.52,E2 -9825.52} C_VEL
LIN {X 0,Y 427.746,Z 425.306,A -85,B 0,C 180,E1 -9826.956,E2 -9826.956} C_VEL
LIN {X 0,Y 428.872,Z 413.134,A -85,B 0,C 180,E1 -9828.388,E2 -9828.388} C_VEL
LIN {X 0,Y 430.056,Z 399.777,A -85,B 0,C 180,E1 -9829.698,E2 -9829.698} C_VEL
LIN {X 0,Y 431.372,Z 385.084,A -85,B 0,C 180,E1 -9830.879,E2 -9830.879} C_VEL
LIN {X 0,Y 432.696,Z 369.567,A -85,B 0,C 180,E1 -9831.874,E2 -9831.874} C_VEL
LIN {X 0,Y 433.469,Z 357.762,A -85,B 0,C 180,E1 -9832.487,E2 -9832.487} C_VEL
LIN {X 0,Y 430.331,Z 342.176,A -85,B 0,C 180,E1 -9833.366,E2 -9833.366} C_VEL
LIN {X 0,Y 426.79,Z 326.236,A -85,B 0,C 180,E1 -9834.133,E2 -9834.133} C_VEL
LIN {X 0,Y 425.318,Z 320.293,A -85,B 0,C 180,E1 -9834.422,E2 -9834.422} C_VEL
LIN {X 0,Y 425.68,Z 312.674,A -85,B 0,C 180,E1 -9837.535,E2 -9837.535} C_VEL
LIN {X 0,Y 426.049,Z 306.453,A -85,B 0,C 180,E1 -9840.207,E2 -9840.207} C_VEL
LIN {X 0,Y 426.548,Z 299.314,A -85,B 0,C 180,E1 -9843.502,E2 -9843.502} C_VEL
LIN {X 0,Y 427.162,Z 292.734,A -85,B 0,C 180,E1 -9846.908,E2 -9846.908} C_VEL
LIN {X 0,Y 427.734,Z 287.893,A -85,B 0,C 180,E1 -9849.852,E2 -9849.852} C_VEL
LIN {X 0,Y 428.109,Z 284.536,A -85,B 0,C 180,E1 -9852.376,E2 -9852.376} C_VEL
LIN {X 0,Y 427.888,Z 282.069,A -85,B 0,C 180,E1 -9854.933,E2 -9854.933} C_VEL
LIN {X 0,Y 427.683,Z 281.08,A -85,B 0,C 180,E1 -9856.356,E2 -9856.356} C_VEL
LIN {X 0,Y 427.034,Z 279.902,A -85,B 0,C 180,E1 -9859.206,E2 -9859.206} C_VEL
LIN {X 0,Y 426.444,Z 279.577,A -85,B 0,C 180,E1 -9862.427,E2 -9862.427} C_VEL
LIN {X 0,Y 425.956,Z 280.152,A -85,B 0,C 180,E1 -9865.877,E2 -9865.877} C_VEL
LIN {X 0,Y 425.624,Z 281.332,A -85,B 0,C 180,E1 -9869.211,E2 -9869.211} C_VEL
LIN {X 0,Y 425.418,Z 282.707,A -85,B 0,C 180,E1 -9872.08,E2 -9872.08} C_VEL
LIN {X 0,Y 426.583,Z 285.74,A -85,B 0,C 180,E1 -9872.288,E2 -9872.288} C_VEL
LIN {X 0,Y 431.607,Z 297.861,A -85,B 0,C 180,E1 -9873.129,E2 -9873.129} C_VEL
LIN {X 0,Y 433.634,Z 304.348,A -85,B 0,C 180,E1 -9873.567,E2 -9873.567} C_VEL
LIN {X 0,Y 433.63,Z 309.586,A -85,B 0,C 180,E1 -9873.829,E2 -9873.829} C_VEL
LIN {X 0,Y 432.667,Z 324.462,A -85,B 0,C 180,E1 -9874.633,E2 -9874.633} C_VEL
LIN {X 0,Y 431.6,Z 339.289,A -85,B 0,C 180,E1 -9875.646,E2 -9875.646} C_VEL
LIN {X 0,Y 430.455,Z 353.104,A -85,B 0,C 180,E1 -9876.806,E2 -9876.806} C_VEL
LIN {X 0,Y 429.396,Z 366.119,A -85,B 0,C 180,E1 -9878.139,E2 -9878.139} C_VEL
LIN {X 0,Y 428.438,Z 376.339,A -85,B 0,C 180,E1 -9879.377,E2 -9879.377} C_VEL
LIN {X 0,Y 427.589,Z 386.381,A -85,B 0,C 180,E1 -9880.809,E2 -9880.809} C_VEL
LIN {X 0,Y 426.619,Z 396.301,A -85,B 0,C 180,E1 -9882.504,E2 -9882.504} C_VEL
LIN {X 0,Y 425.905,Z 404.473,A -85,B 0,C 180,E1 -9884.201,E2 -9884.201} C_VEL
LIN {X 0,Y 425.315,Z 412.032,A -85,B 0,C 180,E1 -9886.137,E2 -9886.137} C_VEL
LIN {X 0,Y 424.885,Z 417.938,A -85,B 0,C 180,E1 -9888.068,E2 -9888.068} C_VEL
LIN {X 0,Y 424.599,Z 421.377,A -85,B 0,C 180,E1 -9889.51,E2 -9889.51} C_VEL
LIN {X 0,Y 424.435,Z 424.775,A -85,B 0,C 180,E1 -9891.43,E2 -9891.43} C_VEL
LIN {X 0,Y 424.361,Z 427.072,A -85,B 0,C 180,E1 -9893.56,E2 -9893.56} C_VEL
LIN {X 0,Y 424.244,Z 427.819,A -85,B 0,C 180,E1 -9895.249,E2 -9895.249} C_VEL
LIN {X 0,Y 424.317,Z 427.522,A -85,B 0,C 180,E1 -9897.152,E2 -9897.152} C_VEL
LIN {X 0,Y 424.257,Z 426.04,A -85,B 0,C 180,E1 -9899.051,E2 -9899.051} C_VEL
LIN {X 0,Y 424.274,Z 423.313,A -85,B 0,C 180,E1 -9900.949,E2 -9900.949} C_VEL
LIN {X 0,Y 424.561,Z 419.308,A -85,B 0,C 180,E1 -9902.847,E2 -9902.847} C_VEL
LIN {X 0,Y 424.946,Z 413.963,A -85,B 0,C 180,E1 -9904.744,E2 -9904.744} C_VEL
LIN {X 0,Y 425.156,Z 409.007,A -85,B 0,C 180,E1 -9906.168,E2 -9906.168} C_VEL
LIN {X 0,Y 425.687,Z 401.169,A -85,B 0,C 180,E1 -9908.02,E2 -9908.02} C_VEL
LIN {X 0,Y 426.356,Z 392.352,A -85,B 0,C 180,E1 -9909.728,E2 -9909.728} C_VEL
LIN {X 0,Y 427.258,Z 382.025,A -85,B 0,C 180,E1 -9911.385,E2 -9911.385} C_VEL
LIN {X 0,Y 428.116,Z 371.498,A -85,B 0,C 180,E1 -9912.804,E2 -9912.804} C_VEL
LIN {X 0,Y 429.02,Z 360.101,A -85,B 0,C 180,E1 -9914.104,E2 -9914.104} C_VEL
LIN {X 0,Y 429.964,Z 347.206,A -85,B 0,C 180,E1 -9915.336,E2 -9915.336} C_VEL
LIN {X 0,Y 430.913,Z 334.538,A -85,B 0,C 180,E1 -9916.34,E2 -9916.34} C_VEL
LIN {X 0,Y 431.807,Z 320.118,A -85,B 0,C 180,E1 -9917.274,E2 -9917.274} C_VEL
LIN {X 0,Y 432.616,Z 304.911,A -85,B 0,C 180,E1 -9918.046,E2 -9918.046} C_VEL
LIN {X 0,Y 432.44,Z 302.685,A -85,B 0,C 180,E1 -9918.152,E2 -9918.152} C_VEL
LIN {X 0,Y 427.823,Z 286.507,A -85,B 0,C 180,E1 -9918.986,E2 -9918.986} C_VEL
LIN {X 0,Y 424.476,Z 275.457,A -85,B 0,C 180,E1 -9919.484,E2 -9919.484} C_VEL
LIN {X 0,Y 424.503,Z 272.657,A -85,B 0,C 180,E1 -9922.383,E2 -9922.383} C_VEL
LIN {X 0,Y 424.576,Z 269.71,A -85,B 0,C 180,E1 -9925.492,E2 -9925.492} C_VEL
LIN {X 0,Y 424.579,Z 267.74,A -85,B 0,C 180,E1 -9927.612,E2 -9927.612} C_VEL
LIN {X 0,Y 424.687,Z 267.212,A -85,B 0,C 180,E1 -9928.707,E2 -9928.707} C_VEL
LIN {X 0,Y 424.999,Z 267.172,A -85,B 0,C 180,E1 -9931.95,E2 -9931.95} C_VEL
LIN {X 0,Y 425.274,Z 267.139,A -85,B 0,C 180,E1 -9935.339,E2 -9935.339} C_VEL
LIN {X 0,Y 425.295,Z 267.136,A -85,B 0,C 180,E1 -9938.899,E2 -9938.899} C_VEL
LIN {X 0,Y 425.286,Z 267.134,A -85,B 0,C 180,E1 -9941.957,E2 -9941.957} C_VEL
LIN {X 0,Y 425.288,Z 267.135,A -85,B 0,C 180,E1 -9945.283,E2 -9945.283} C_VEL
LIN {X 0,Y 425.278,Z 267.136,A -85,B 0,C 180,E1 -9948.621,E2 -9948.621} C_VEL
LIN {X 0,Y 425.305,Z 267.133,A -85,B 0,C 180,E1 -9951.102,E2 -9951.102} C_VEL
LIN {X 0,Y 425.301,Z 267.134,A -85,B 0,C 180,E1 -9954.664,E2 -9954.664} C_VEL
LIN {X 0,Y 425.268,Z 267.136,A -85,B 0,C 180,E1 -9958.073,E2 -9958.073} C_VEL
LIN {X 0,Y 425.334,Z 267.129,A -85,B 0,C 180,E1 -9961.368,E2 -9961.368} C_VEL
LIN {X 0,Y 425.286,Z 267.137,A -85,B 0,C 180,E1 -9964.554,E2 -9964.554} C_VEL
LIN {X 0,Y 425.286,Z 267.135,A -85,B 0,C 180,E1 -9966.634,E2 -9966.634} C_VEL
LIN {X 0,Y 425.298,Z 267.133,A -85,B 0,C 180,E1 -9969.695,E2 -9969.695} C_VEL
LIN {X 0,Y 425.342,Z 267.128,A -85,B 0,C 180,E1 -9972.697,E2 -9972.697} C_VEL
LIN {X 0,Y 425.35,Z 267.127,A -85,B 0,C 180,E1 -9975.65,E2 -9975.65} C_VEL
LIN {X 0,Y 425.353,Z 267.126,A -85,B 0,C 180,E1 -9978.564,E2 -9978.564} C_VEL
LIN {X 0,Y 425.44,Z 267.116,A -85,B 0,C 180,E1 -9981.45,E2 -9981.45} C_VEL
LIN {X 0,Y 425.531,Z 267.106,A -85,B 0,C 180,E1 -9984.313,E2 -9984.313} C_VEL
LIN {X 0,Y 425.576,Z 267.1,A -85,B 0,C 180,E1 -9988.107,E2 -9988.107} C_VEL
LIN {X 0,Y 425.7,Z 267.085,A -85,B 0,C 180,E1 -9990,E2 -9990} C_VEL
LIN {X 0,Y 425.541,Z 267.101,A -85,B 0,C 180,E1 -9992.84,E2 -9992.84} C_VEL
LIN {X 0,Y 425.412,Z 267.117,A -85,B 0,C 180,E1 -9993.336,E2 -9993.336} C_VEL
LIN {X 0,Y 424.639,Z 267.217,A -85,B 0,C 180,E1 -9994.127,E2 -9994.127} C_VEL
LIN {X 0,Y 421.802,Z 267.57,A -85,B 0,C 180,E1 -9995.413,E2 -9995.413} C_VEL
LIN {X 0,Y 419.485,Z 267.857,A -85,B 0,C 180,E1 -9996.452,E2 -9996.452} C_VEL
LIN {X 0,Y 418.514,Z 267.978,A -85,B 0,C 180,E1 -9997.253,E2 -9997.253} C_VEL
LIN {X 0,Y 418.442,Z 267.987,A -85,B 0,C 180,E1 -9997.524,E2 -9997.524} C_VEL
LIN {X 0,Y 418.335,Z 268,A -85,B 0,C 180,E1 -10000.65,E2 -10000.65} C_VEL
LIN {X 0,Y 418.316,Z 268.004,A -85,B 0,C 180,E1 -10003.604,E2 -10003.604} C_VEL
LIN {X 0,Y 418.316,Z 268.001,A -85,B 0,C 180,E1 -10006.735,E2 -10006.735} C_VEL
LIN {X 0,Y 418.274,Z 268.01,A -85,B 0,C 180,E1 -10009.79,E2 -10009.79} C_VEL
LIN {X 0,Y 418.242,Z 268.01,A -85,B 0,C 180,E1 -10012.736,E2 -10012.736} C_VEL
LIN {X 0,Y 418.274,Z 268.009,A -85,B 0,C 180,E1 -10015.904,E2 -10015.904} C_VEL
LIN {X 0,Y 418.268,Z 268.01,A -85,B 0,C 180,E1 -10019.162,E2 -10019.162} C_VEL
LIN {X 0,Y 418.261,Z 268.011,A -85,B 0,C 180,E1 -10022.844,E2 -10022.844} C_VEL
LIN {X 0,Y 418.247,Z 268.009,A -85,B 0,C 180,E1 -10026.238,E2 -10026.238} C_VEL
LIN {X 0,Y 418.212,Z 268.017,A -85,B 0,C 180,E1 -10029.687,E2 -10029.687} C_VEL
LIN {X 0,Y 418.212,Z 268.015,A -85,B 0,C 180,E1 -10032.318,E2 -10032.318} C_VEL
LIN {X 0,Y 418.239,Z 268.013,A -85,B 0,C 180,E1 -10035.109,E2 -10035.109} C_VEL
LIN {X 0,Y 418.244,Z 268.011,A -85,B 0,C 180,E1 -10037.767,E2 -10037.767} C_VEL
LIN {X 0,Y 418.259,Z 268.012,A -85,B 0,C 180,E1 -10040.619,E2 -10040.619} C_VEL
LIN {X 0,Y 418.246,Z 268.011,A -85,B 0,C 180,E1 -10043.976,E2 -10043.976} C_VEL
LIN {X 0,Y 418.261,Z 268.009,A -85,B 0,C 180,E1 -10047.156,E2 -10047.156} C_VEL
LIN {X 0,Y 418.273,Z 268.01,A -85,B 0,C 180,E1 -10050.895,E2 -10050.895} C_VEL
LIN {X 0,Y 418.266,Z 268.008,A -85,B 0,C 180,E1 -10054.095,E2 -10054.095} C_VEL
LIN {X 0,Y 418.236,Z 268.013,A -85,B 0,C 180,E1 -10057.263,E2 -10057.263} C_VEL
LIN {X 0,Y 418.287,Z 268.009,A -85,B 0,C 180,E1 -10060.364,E2 -10060.364} C_VEL
LIN {X 0,Y 418.321,Z 268.002,A -85,B 0,C 180,E1 -10063.405,E2 -10063.405} C_VEL
LIN {X 0,Y 418.351,Z 267.996,A -85,B 0,C 180,E1 -10066.999,E2 -10066.999} C_VEL
LIN {X 0,Y 418.344,Z 268.001,A -85,B 0,C 180,E1 -10070.328,E2 -10070.328} C_VEL
LIN {X 0,Y 418.446,Z 267.985,A -85,B 0,C 180,E1 -10073.248,E2 -10073.248} C_VEL
LIN {X 0,Y 418.331,Z 267.999,A -85,B 0,C 180,E1 -10075.181,E2 -10075.181} C_VEL
LIN {X 0,Y 418.546,Z 267.975,A -85,B 0,C 180,E1 -10078.075,E2 -10078.075} C_VEL
LIN {X 0,Y 418.669,Z 267.961,A -85,B 0,C 180,E1 -10080,E2 -10080} C_VEL
LIN {X 0,Y 418.505,Z 267.978,A -85,B 0,C 180,E1 -10082.888,E2 -10082.888} C_VEL
LIN {X 0,Y 418.497,Z 267.981,A -85,B 0,C 180,E1 -10085.783,E2 -10085.783} C_VEL
LIN {X 0,Y 418.38,Z 267.993,A -85,B 0,C 180,E1 -10088.695,E2 -10088.695} C_VEL
LIN {X 0,Y 418.319,Z 268.004,A -85,B 0,C 180,E1 -10091.631,E2 -10091.631} C_VEL
LIN {X 0,Y 418.305,Z 268.002,A -85,B 0,C 180,E1 -10094.597,E2 -10094.597} C_VEL
LIN {X 0,Y 418.289,Z 268.007,A -85,B 0,C 180,E1 -10097.603,E2 -10097.603} C_VEL
LIN {X 0,Y 418.253,Z 268.009,A -85,B 0,C 180,E1 -10100.663,E2 -10100.663} C_VEL
LIN {X 0,Y 418.288,Z 268.007,A -85,B 0,C 180,E1 -10103.781,E2 -10103.781} C_VEL
LIN {X 0,Y 418.225,Z 268.014,A -85,B 0,C 180,E1 -10107.046,E2 -10107.046} C_VEL
LIN {X 0,Y 418.243,Z 268.012,A -85,B 0,C 180,E1 -10110.272,E2 -10110.272} C_VEL
LIN {X 0,Y 418.25,Z 268.013,A -85,B 0,C 180,E1 -10113.677,E2 -10113.677} C_VEL
LIN {X 0,Y 418.241,Z 268.009,A -85,B 0,C 180,E1 -10117.224,E2 -10117.224} C_VEL
LIN {X 0,Y 418.253,Z 268.067,A -85,B 0,C 180,E1 -10117.543,E2 -10117.543} C_VEL
LIN {X 0,Y 419.221,Z 273.519,A -85,B 0,C 180,E1 -10121.027,E2 -10121.027} C_VEL
LIN {X 0,Y 420.156,Z 278.464,A -85,B 0,C 180,E1 -10124.006,E2 -10124.006} C_VEL
LIN {X 0,Y 421.027,Z 283.385,A -85,B 0,C 180,E1 -10126.812,E2 -10126.812} C_VEL
LIN {X 0,Y 421.192,Z 286.858,A -85,B 0,C 180,E1 -10128.665,E2 -10128.665} C_VEL
LIN {X 0,Y 420.7,Z 293.134,A -85,B 0,C 180,E1 -10131.822,E2 -10131.822} C_VEL
LIN {X 0,Y 420.113,Z 299.856,A -85,B 0,C 180,E1 -10135.056,E2 -10135.056} C_VEL
LIN {X 0,Y 419.489,Z 307.765,A -85,B 0,C 180,E1 -10138.71,E2 -10138.71} C_VEL
LIN {X 0,Y 419.078,Z 313.891,A -85,B 0,C 180,E1 -10141.448,E2 -10141.448} C_VEL
LIN {X 0,Y 418.58,Z 321.242,A -85,B 0,C 180,E1 -10144.643,E2 -10144.643} C_VEL
LIN {X 0,Y 418.499,Z 323.123,A -85,B 0,C 180,E1 -10145.397,E2 -10145.397} C_VEL
LIN {X 0,Y 422.949,Z 340.157,A -85,B 0,C 180,E1 -10146.136,E2 -10146.136} C_VEL
LIN {X 0,Y 426.391,Z 355.707,A -85,B 0,C 180,E1 -10146.962,E2 -10146.962} C_VEL
LIN {X 0,Y 426.973,Z 359.618,A -85,B 0,C 180,E1 -10147.185,E2 -10147.185} C_VEL
LIN {X 0,Y 425.974,Z 373.987,A -85,B 0,C 180,E1 -10147.954,E2 -10147.954} C_VEL
LIN {X 0,Y 424.664,Z 388.088,A -85,B 0,C 180,E1 -10148.902,E2 -10148.902} C_VEL
LIN {X 0,Y 423.463,Z 401.07,A -85,B 0,C 180,E1 -10149.983,E2 -10149.983} C_VEL
LIN {X 0,Y 422.143,Z 414.197,A -85,B 0,C 180,E1 -10151.308,E2 -10151.308} C_VEL
LIN {X 0,Y 420.994,Z 426.145,A -85,B 0,C 180,E1 -10152.763,E2 -10152.763} C_VEL
LIN {X 0,Y 419.982,Z 436.234,A -85,B 0,C 180,E1 -10154.221,E2 -10154.221} C_VEL
LIN {X 0,Y 418.978,Z 446.12,A -85,B 0,C 180,E1 -10155.923,E2 -10155.923} C_VEL
LIN {X 0,Y 418.331,Z 454.368,A -85,B 0,C 180,E1 -10157.631,E2 -10157.631} C_VEL
LIN {X 0,Y 417.773,Z 461.212,A -85,B 0,C 180,E1 -10159.336,E2 -10159.336} C_VEL
LIN {X 0,Y 417.396,Z 467.544,A -85,B 0,C 180,E1 -10161.284,E2 -10161.284} C_VEL
LIN {X 0,Y 417.169,Z 472.442,A -85,B 0,C 180,E1 -10163.227,E2 -10163.227} C_VEL
LIN {X 0,Y 417.088,Z 476.029,A -85,B 0,C 180,E1 -10165.167,E2 -10165.167} C_VEL
LIN {X 0,Y 417.07,Z 478.378,A -85,B 0,C 180,E1 -10167.102,E2 -10167.102} C_VEL
LIN {X 0,Y 416.989,Z 479.537,A -85,B 0,C 180,E1 -10169.034,E2 -10169.034} C_VEL
LIN {X 0,Y 416.989,Z 479.493,A -85,B 0,C 180,E1 -10170.966,E2 -10170.966} C_VEL
LIN {X 0,Y 417.085,Z 478.254,A -85,B 0,C 180,E1 -10172.898,E2 -10172.898} C_VEL
LIN {X 0,Y 417.096,Z 475.815,A -85,B 0,C 180,E1 -10174.833,E2 -10174.833} C_VEL
LIN {X 0,Y 417.226,Z 472.131,A -85,B 0,C 180,E1 -10176.772,E2 -10176.772} C_VEL
LIN {X 0,Y 417.396,Z 467.1,A -85,B 0,C 180,E1 -10178.716,E2 -10178.716} C_VEL
LIN {X 0,Y 417.773,Z 460.595,A -85,B 0,C 180,E1 -10180.664,E2 -10180.664} C_VEL
LIN {X 0,Y 418.315,Z 453.584,A -85,B 0,C 180,E1 -10182.369,E2 -10182.369} C_VEL
LIN {X 0,Y 418.93,Z 445.117,A -85,B 0,C 180,E1 -10184.079,E2 -10184.079} C_VEL
LIN {X 0,Y 419.879,Z 434.998,A -85,B 0,C 180,E1 -10185.783,E2 -10185.783} C_VEL
LIN {X 0,Y 421.018,Z 422.813,A -85,B 0,C 180,E1 -10187.486,E2 -10187.486} C_VEL
LIN {X 0,Y 422.22,Z 410.287,A -85,B 0,C 180,E1 -10188.941,E2 -10188.941} C_VEL
LIN {X 0,Y 423.489,Z 397.913,A -85,B 0,C 180,E1 -10190.143,E2 -10190.143} C_VEL
LIN {X 0,Y 424.704,Z 384.64,A -85,B 0,C 180,E1 -10191.222,E2 -10191.222} C_VEL
LIN {X 0,Y 426.089,Z 369.34,A -85,B 0,C 180,E1 -10192.231,E2 -10192.231} C_VEL
LIN {X 0,Y 426.772,Z 358.23,A -85,B 0,C 180,E1 -10192.835,E2 -10192.835} C_VEL
LIN {X 0,Y 423.167,Z 339.98,A -85,B 0,C 180,E1 -10193.917,E2 -10193.917} C_VEL
LIN {X 0,Y 419.927,Z 325.95,A -85,B 0,C 180,E1 -10194.636,E2 -10194.636} C_VEL
LIN {X 0,Y 418.331,Z 319.612,A -85,B 0,C 180,E1 -10194.954,E2 -10194.954} C_VEL
LIN {X 0,Y 418.696,Z 312.317,A -85,B 0,C 180,E1 -10198.034,E2 -10198.034} C_VEL
LIN {X 0,Y 419.056,Z 306.291,A -85,B 0,C 180,E1 -10200.717,E2 -10200.717} C_VEL
LIN {X 0,Y 419.592,Z 299.196,A -85,B 0,C 180,E1 -10204.133,E2 -10204.133} C_VEL
LIN {X 0,Y 420.187,Z 293.827,A -85,B 0,C 180,E1 -10207.023,E2 -10207.023} C_VEL
LIN {X 0,Y 420.759,Z 289.388,A -85,B 0,C 180,E1 -10209.795,E2 -10209.795} C_VEL
LIN {X 0,Y 421.079,Z 286.6,A -85,B 0,C 180,E1 -10211.884,E2 -10211.884} C_VEL
LIN {X 0,Y 421.038,Z 284.256,A -85,B 0,C 180,E1 -10214.13,E2 -10214.13} C_VEL
LIN {X 0,Y 420.655,Z 282.362,A -85,B 0,C 180,E1 -10216.765,E2 -10216.765} C_VEL
LIN {X 0,Y 420.097,Z 281.367,A -85,B 0,C 180,E1 -10219.274,E2 -10219.274} C_VEL
LIN {X 0,Y 419.588,Z 281.001,A -85,B 0,C 180,E1 -10221.929,E2 -10221.929} C_VEL
LIN {X 0,Y 419.063,Z 281.353,A -85,B 0,C 180,E1 -10225.263,E2 -10225.263} C_VEL
LIN {X 0,Y 418.805,Z 281.97,A -85,B 0,C 180,E1 -10227.521,E2 -10227.521} C_VEL
LIN {X 0,Y 418.483,Z 283.313,A -85,B 0,C 180,E1 -10230.855,E2 -10230.855} C_VEL
LIN {X 0,Y 418.438,Z 283.635,A -85,B 0,C 180,E1 -10231.525,E2 -10231.525} C_VEL
LIN {X 0,Y 419.607,Z 286.625,A -85,B 0,C 180,E1 -10231.75,E2 -10231.75} C_VEL
LIN {X 0,Y 424.795,Z 298.559,A -85,B 0,C 180,E1 -10232.652,E2 -10232.652} C_VEL
LIN {X 0,Y 427.384,Z 306.695,A -85,B 0,C 180,E1 -10233.237,E2 -10233.237} C_VEL
LIN {X 0,Y 426.523,Z 321.78,A -85,B 0,C 180,E1 -10234.044,E2 -10234.044} C_VEL
LIN {X 0,Y 425.284,Z 337.287,A -85,B 0,C 180,E1 -10235.078,E2 -10235.078} C_VEL
LIN {X 0,Y 424.13,Z 351.03,A -85,B 0,C 180,E1 -10236.21,E2 -10236.21} C_VEL
LIN {X 0,Y 422.931,Z 364.195,A -85,B 0,C 180,E1 -10237.53,E2 -10237.53} C_VEL
LIN {X 0,Y 421.87,Z 375.585,A -85,B 0,C 180,E1 -10238.895,E2 -10238.895} C_VEL
LIN {X 0,Y 420.806,Z 386.686,A -85,B 0,C 180,E1 -10240.487,E2 -10240.487} C_VEL
LIN {X 0,Y 419.771,Z 396.647,A -85,B 0,C 180,E1 -10242.209,E2 -10242.209} C_VEL
LIN {X 0,Y 419.021,Z 404.866,A -85,B 0,C 180,E1 -10243.934,E2 -10243.934} C_VEL
LIN {X 0,Y 418.355,Z 412.435,A -85,B 0,C 180,E1 -10245.902,E2 -10245.902} C_VEL
LIN {X 0,Y 417.892,Z 418.365,A -85,B 0,C 180,E1 -10247.865,E2 -10247.865} C_VEL
LIN {X 0,Y 417.575,Z 421.823,A -85,B 0,C 180,E1 -10249.331,E2 -10249.331} C_VEL
LIN {X 0,Y 417.369,Z 425.246,A -85,B 0,C 180,E1 -10251.283,E2 -10251.283} C_VEL
LIN {X 0,Y 417.306,Z 427.383,A -85,B 0,C 180,E1 -10253.23,E2 -10253.23} C_VEL
LIN {X 0,Y 417.177,Z 428.306,A -85,B 0,C 180,E1 -10255.168,E2 -10255.168} C_VEL
LIN {X 0,Y 417.249,Z 428.019,A -85,B 0,C 180,E1 -10257.104,E2 -10257.104} C_VEL
LIN {X 0,Y 417.201,Z 426.533,A -85,B 0,C 180,E1 -10259.035,E2 -10259.035} C_VEL
LIN {X 0,Y 417.219,Z 423.798,A -85,B 0,C 180,E1 -10260.965,E2 -10260.965} C_VEL
LIN {X 0,Y 417.49,Z 419.786,A -85,B 0,C 180,E1 -10262.895,E2 -10262.895} C_VEL
LIN {X 0,Y 417.908,Z 414.425,A -85,B 0,C 180,E1 -10264.824,E2 -10264.824} C_VEL
LIN {X 0,Y 418.147,Z 407.606,A -85,B 0,C 180,E1 -10266.757,E2 -10266.757} C_VEL
LIN {X 0,Y 418.795,Z 400.348,A -85,B 0,C 180,E1 -10268.42,E2 -10268.42} C_VEL
LIN {X 0,Y 419.544,Z 391.389,A -85,B 0,C 180,E1 -10270.131,E2 -10270.131} C_VEL
LIN {X 0,Y 420.304,Z 382.421,A -85,B 0,C 180,E1 -10271.576,E2 -10271.576} C_VEL
LIN {X 0,Y 421.222,Z 371.873,A -85,B 0,C 180,E1 -10273.018,E2 -10273.018} C_VEL
LIN {X 0,Y 422.293,Z 359.291,A -85,B 0,C 180,E1 -10274.456,E2 -10274.456} C_VEL
LIN {X 0,Y 423.174,Z 346.772,A -85,B 0,C 180,E1 -10275.657,E2 -10275.657} C_VEL
LIN {X 0,Y 424.253,Z 333.178,A -85,B 0,C 180,E1 -10276.728,E2 -10276.728} C_VEL
LIN {X 0,Y 425.181,Z 318.525,A -85,B 0,C 180,E1 -10277.665,E2 -10277.665} C_VEL
LIN {X 0,Y 425.82,Z 304.78,A -85,B 0,C 180,E1 -10278.368,E2 -10278.368} C_VEL
LIN {X 0,Y 421.491,Z 289.274,A -85,B 0,C 180,E1 -10279.208,E2 -10279.208} C_VEL
LIN {X 0,Y 417.428,Z 275.846,A -85,B 0,C 180,E1 -10279.829,E2 -10279.829} C_VEL
LIN {X 0,Y 417.447,Z 273.001,A -85,B 0,C 180,E1 -10282.782,E2 -10282.782} C_VEL
LIN {X 0,Y 417.516,Z 270.997,A -85,B 0,C 180,E1 -10284.887,E2 -10284.887} C_VEL
LIN {X 0,Y 417.534,Z 268.104,A -85,B 0,C 180,E1 -10288.119,E2 -10288.119} C_VEL
LIN {X 0,Y 417.886,Z 268.06,A -85,B 0,C 180,E1 -10291.424,E2 -10291.424} C_VEL
LIN {X 0,Y 418.177,Z 268.021,A -85,B 0,C 180,E1 -10294.562,E2 -10294.562} C_VEL
LIN {X 0,Y 418.241,Z 268.014,A -85,B 0,C 180,E1 -10297.224,E2 -10297.224} C_VEL
LIN {X 0,Y 418.245,Z 268.012,A -85,B 0,C 180,E1 -10299.683,E2 -10299.683} C_VEL
LIN {X 0,Y 418.227,Z 268.014,A -85,B 0,C 180,E1 -10302.32,E2 -10302.32} C_VEL
LIN {X 0,Y 418.239,Z 268.013,A -85,B 0,C 180,E1 -10305.109,E2 -10305.109} C_VEL
LIN {X 0,Y 418.243,Z 268.011,A -85,B 0,C 180,E1 -10307.767,E2 -10307.767} C_VEL
LIN {X 0,Y 418.252,Z 268.012,A -85,B 0,C 180,E1 -10310.62,E2 -10310.62} C_VEL
LIN {X 0,Y 418.246,Z 268.011,A -85,B 0,C 180,E1 -10313.976,E2 -10313.976} C_VEL
LIN {X 0,Y 418.26,Z 268.009,A -85,B 0,C 180,E1 -10317.156,E2 -10317.156} C_VEL
LIN {X 0,Y 418.272,Z 268.01,A -85,B 0,C 180,E1 -10320.895,E2 -10320.895} C_VEL
LIN {X 0,Y 418.264,Z 268.009,A -85,B 0,C 180,E1 -10324.095,E2 -10324.095} C_VEL
LIN {X 0,Y 418.234,Z 268.013,A -85,B 0,C 180,E1 -10327.263,E2 -10327.263} C_VEL
LIN {X 0,Y 418.286,Z 268.009,A -85,B 0,C 180,E1 -10330.364,E2 -10330.364} C_VEL
LIN {X 0,Y 418.32,Z 268.002,A -85,B 0,C 180,E1 -10333.405,E2 -10333.405} C_VEL
LIN {X 0,Y 418.35,Z 267.997,A -85,B 0,C 180,E1 -10336.999,E2 -10336.999} C_VEL
LIN {X 0,Y 418.343,Z 268,A -85,B 0,C 180,E1 -10340.329,E2 -10340.329} C_VEL
LIN {X 0,Y 418.446,Z 267.986,A -85,B 0,C 180,E1 -10343.248,E2 -10343.248} C_VEL
LIN {X 0,Y 418.329,Z 267.999,A -85,B 0,C 180,E1 -10345.181,E2 -10345.181} C_VEL
LIN {X 0,Y 418.544,Z 267.976,A -85,B 0,C 180,E1 -10348.075,E2 -10348.075} C_VEL
LIN {X 0,Y 418.67,Z 267.961,A -85,B 0,C 180,E1 -10350,E2 -10350} C_VEL
LIN {X 0,Y 418.496,Z 267.979,A -85,B 0,C 180,E1 -10352.888,E2 -10352.888} C_VEL
LIN {X 0,Y 418.502,Z 267.981,A -85,B 0,C 180,E1 -10355.783,E2 -10355.783} C_VEL
LIN {X 0,Y 418.442,Z 267.987,A -85,B 0,C 180,E1 -10357.524,E2 -10357.524} C_VEL
LIN {X 0,Y 417.774,Z 268.074,A -85,B 0,C 180,E1 -10358.327,E2 -10358.327} C_VEL
LIN {X 0,Y 414.853,Z 268.437,A -85,B 0,C 180,E1 -10359.629,E2 -10359.629} C_VEL
LIN {X 0,Y 412.387,Z 268.74,A -85,B 0,C 180,E1 -10360.681,E2 -10360.681} C_VEL
LIN {X 0,Y 411.353,Z 268.872,A -85,B 0,C 180,E1 -10361.496,E2 -10361.496} C_VEL
LIN {X 0,Y 411.283,Z 268.88,A -85,B 0,C 180,E1 -10361.772,E2 -10361.772} C_VEL
LIN {X 0,Y 411.262,Z 268.88,A -85,B 0,C 180,E1 -10364.853,E2 -10364.853} C_VEL
LIN {X 0,Y 411.249,Z 268.884,A -85,B 0,C 180,E1 -10367.915,E2 -10367.915} C_VEL
LIN {X 0,Y 411.2,Z 268.889,A -85,B 0,C 180,E1 -10371.034,E2 -10371.034} C_VEL
LIN {X 0,Y 411.231,Z 268.885,A -85,B 0,C 180,E1 -10374.215,E2 -10374.215} C_VEL
LIN {X 0,Y 411.262,Z 268.884,A -85,B 0,C 180,E1 -10377.478,E2 -10377.478} C_VEL
LIN {X 0,Y 411.193,Z 268.891,A -85,B 0,C 180,E1 -10380.848,E2 -10380.848} C_VEL
LIN {X 0,Y 411.209,Z 268.887,A -85,B 0,C 180,E1 -10384.334,E2 -10384.334} C_VEL
LIN {X 0,Y 411.189,Z 268.89,A -85,B 0,C 180,E1 -10387.975,E2 -10387.975} C_VEL
LIN {X 0,Y 411.153,Z 268.898,A -85,B 0,C 180,E1 -10391.226,E2 -10391.226} C_VEL
LIN {X 0,Y 411.177,Z 268.892,A -85,B 0,C 180,E1 -10394.491,E2 -10394.491} C_VEL
LIN {X 0,Y 411.181,Z 268.891,A -85,B 0,C 180,E1 -10398.195,E2 -10398.195} C_VEL
LIN {X 0,Y 411.224,Z 268.889,A -85,B 0,C 180,E1 -10400.776,E2 -10400.776} C_VEL
